// TwinCAT 3 PLC project PLC_
// ProgramVersion: 3.1.4026.24
// libraries:
//   Tc2_EtherCAT, * (Beckhoff Automation GmbH)
//   Tc2_MC2, * (Beckhoff Automation GmbH)
//   Tc2_Standard, * (Beckhoff Automation GmbH)
//   Tc2_SUPS, * (Beckhoff Automation GmbH)
//   Tc2_System, * (Beckhoff Automation GmbH)
//   Tc2_Utilities, * (Beckhoff Automation GmbH)
//   Tc3_McCollisionAvoidance, * (Beckhoff Automation GmbH)
//   Tc3_McCoordinatedMotion, * (Beckhoff Automation GmbH)
//   Tc3_Module, * (Beckhoff Automation GmbH)
// project tree:
//   00_GVLs/ HardwareIO.TcGVL, Parameter_PERSISTENT.TcGVL, GVL.TcGVL, HMI_Mapp.TcGVL
//   01_POUs/ Automatic_POU.TcPOU, Initial_POU.TcPOU, MAIN.TcPOU
//   01_POUs/static/ Device_POU.TcPOU, prgInputMapp.TcPOU, Recipe_POU.TcPOU, Manual_POU.TcPOU, MST_POU.TcPOU, UPS_POU.TcPOU
//   02_Unit/01_Customization/ Ass_DualServo.TcPOU, Ass_LoadPic.TcPOU, Ass_Openbox.TcPOU, Ass_Pallet.TcPOU, Ass_RBStack.TcPOU, Ass_Sealing.TcPOU, Ass_StackComv.TcPOU, Ass_UnloadNG.TcPOU, FB_RollRightAngle.TcPOU, ITF_AutoStructCommand.TcIO, MainControl.TcPOU, ST_HMIitfStructCommandTester.TcDUT, ST_Parameter.TcDUT, ST_SlotData.TcDUT
//   02_Unit/03_Axis/ AXIS_REF_Ext.TcPOU, FB_AxisGeneral.TcPOU, ST_HMIAxieControl.TcDUT, FB_ORG_PositiveEndLessByTouchprobe.TcPOU
//   02_Unit/04_Kuka/ E_KR_AutoExtState.TcDUT, E_CS_Status.TcDUT, RB_KR_PickPlace.TcPOU, RB_KR_Stacking.TcPOU, ST_CS_PickIO.TcDUT, ST_KR_sysIO.TcDUT, ST_KR_stackingIO.TcDUT, ST_CS_sysIO.TcDUT
//   02_Unit/99_Other/ FB_EL3356_0010.TcPOU, FB_RecordValue.TcPOU, F_TrimRightSpace.TcPOU, ST_Inventer.TcDUT, ST_InventerUD.TcDUT, Spacil_FC.TcPOU, ST_Operation.TcDUT
//   02_Unit/00_Alarm/ E_Alarm.TcDUT, E_Warn.TcDUT, ST_AlarmFlag.TcDUT, ST_AlarmItem.TcDUT, U_Alarm.TcDUT
//   / GlobalTextList.TcGTLO, LowTask.TcTTO, PlcTask.TcTTO, RecipeManager.TcRMO (not stored)
//   02_Unit/02_Cylinder kit/ E_CylFault.TcTLEO, E_CylinderType.TcTLEO, FB_CylinderBase.TcPOU, ST_Cylinder.TcDUT, ST_CylinderParameter.TcDUT
//   02_Unit/11_EventLogger/ EventLogger.TcPOU, E_EventType.TcTLEO, ST_Event.TcDUT, UpdateEventTimeWithSystemTime.TcPOU
// real-time tasks:
//   TASK PlcTask: cycle T#1ms, priority 20, ADS port 350
//   TASK Job Task: cycle default, priority 32
//   TASK EipTask: cycle T#10ms, priority 1, ADS port 301
//   TASK LowTask: cycle T#10ms, priority 2, ADS port 351
// motion (NC):
//   TASK NC-Task 1 SAF: cycle T#1ms, priority 4, ADS port 501
//   TASK NC-Task 1 SVB: cycle T#2ms, priority 8, ADS port 511
//   AXIS Axis DualServo1 2 (id 1)
//     Dynamic: Acceleration=70000.1, Deceleration=70000.1, Jerk=1633330
//     Velo: Maximum=4000
//     OtherSettings: AllowMotionCmdToSlave=true
//     encoder EncType=19
//       EncPara: ScaleFactorNumerator=91.44, ScaleFactorDenominator=8388608, ModuloFactor=3657.5, Inverse=true, MaxCount=#xffffffff
//         ActPosCorrection: Enable=true, Time=0.1
//     drive DrvType=16
//       DrvPara: Inverse=true, MaxCount=#xffffffff, DriveControlDWord=#x00020100
//         Analog: VeloReferenz=4000, TorqueSetpointScale=10, ScaleFactorActTorque=0.1
//         TimeComp: TaskDelayCycles=1
//     controller CtrType=1
//       CtrPara: PriorControlFactor=1
//         PosDiffControl: Enable=false
//         Observer: BandWidth=20
//   AXIS Axis DualServo2 3 (id 2)
//     Dynamic: Acceleration=70000.1, Deceleration=70000.1, Jerk=1633330
//     Velo: Maximum=4000
//     OtherSettings: AllowMotionCmdToSlave=true
//     encoder EncType=19
//       EncPara: ScaleFactorNumerator=91.44, ScaleFactorDenominator=8388608, ModuloFactor=3657.5, Inverse=true, MaxCount=#xffffffff
//         ActPosCorrection: Enable=true, Time=0.1
//     drive DrvType=16
//       DrvPara: Inverse=true, MaxCount=#xffffffff, DriveControlDWord=#x00020100
//         Analog: VeloReferenz=4000, TorqueSetpointScale=10, ScaleFactorActTorque=0.1
//         TimeComp: TaskDelayCycles=1
//     controller CtrType=1
//       CtrPara: PriorControlFactor=1
//         PosDiffControl: Enable=false
//         Observer: BandWidth=20
//   AXIS Axis_FlyIn 1 (id 3)
//     Dynamic: Acceleration=28000, Deceleration=28000, Jerk=653333
//     Velo: Maximum=1600
//     PositionAreaControl: Enable=false
//     TargetPosControl: Enable=false
//     OtherSettings: AllowMotionCmdToSlave=true
//     encoder EncType=19
//       EncPara: ScaleFactorNumerator=31.9024, ScaleFactorDenominator=8388608, Inverse=true, MaxCount=#xffffffff
//     drive DrvType=16
//       DrvPara: Inverse=true, MaxCount=#xffffffff, DriveControlDWord=#x00020100
//         Analog: TorqueSetpointScale=10, ScaleFactorActTorque=0.1
//         TimeComp: TaskDelayCycles=1
//     controller CtrType=1
//       CtrPara: PriorControlFactor=1
//         PosDiffControl: Enable=false
//         Observer: BandWidth=20
//   AXIS Axis BoxPullout 4 (id 4)
//     Dynamic: Acceleration=12750, Deceleration=12750, Jerk=154821
//     Velo: FastManual=300, Maximum=1500
//     OtherSettings: AllowMotionCmdToSlave=true
//     encoder EncType=19
//       EncPara: ScaleFactorNumerator=6.2831853, ScaleFactorDenominator=8388608, Inverse=true, MaxCount=#xffffffff
//     drive DrvType=16
//       DrvPara: Inverse=true, MaxCount=#xffffffff, DriveControlDWord=#x00020100
//         Analog: VeloReferenz=1500, TorqueSetpointScale=10, ScaleFactorActTorque=0.1
//         TimeComp: TaskDelayCycles=1
//     controller CtrType=1
//       CtrPara: PriorControlFactor=1
//         Observer: BandWidth=20
//   AXIS Axis load1 5 (id 5)
//     Dynamic: Acceleration=12000, Deceleration=12000, Jerk=90000
//     Velo: RefSearch=300, RefSync=300
//     OtherSettings: AllowMotionCmdToSlave=true
//     encoder EncType=19
//       EncPara: ScaleFactorNumerator=31.41599265359, ScaleFactorDenominator=8388608, ModuloFactor=1005, MaxCount=#xffffffff
//         Inc: RefSearchInverse=true, RefSyncInverse=false
//     drive DrvType=16
//       DrvPara: MaxCount=#xffffffff, DriveControlDWord=#x00020100
//         Analog: TorqueSetpointScale=10, ScaleFactorActTorque=0.1
//         TimeComp: TaskDelayCycles=1
//     controller CtrType=1
//       CtrPara: PriorControlFactor=1
//         PosDiffControl: Enable=false
//         Observer: BandWidth=20
//   AXIS Axis load2 6 (id 6)
//     Dynamic: Acceleration=12000, Deceleration=12000, Jerk=90000
//     Velo: RefSearch=300, RefSync=300
//     OtherSettings: AllowMotionCmdToSlave=true
//     encoder EncType=19
//       EncPara: ScaleFactorNumerator=31.41599265359, ScaleFactorDenominator=8388608, ModuloFactor=1005, Inverse=true, MaxCount=#xffffffff
//         Inc: RefSearchInverse=true, RefSyncInverse=false
//     drive DrvType=16
//       DrvPara: Inverse=true, MaxCount=#xffffffff, DriveControlDWord=#x00020100
//         Analog: TorqueSetpointScale=10, ScaleFactorActTorque=0.1
//         TimeComp: TaskDelayCycles=1
//     controller CtrType=1
//       CtrPara: PriorControlFactor=1
//         PosDiffControl: Enable=false
//         Observer: BandWidth=20
// I/O:
//   DEVICE Device 1 (EtherCAT), AmsNetId 10.200.96.23.2.1
//     Term 1 (EK1200) [EK1200-5000 EtherCAT Power supply (2A E-Bus)]
//       Term 2 (EL1889) [EL1889 16Ch. Dig. Input 24V, 3ms, negative]
//       Term 3 (EL1889) [EL1889 16Ch. Dig. Input 24V, 3ms, negative]
//       Term 4 (EL1889) [EL1889 16Ch. Dig. Input 24V, 3ms, negative]
//       Term 5 (EL1889) [EL1889 16Ch. Dig. Input 24V, 3ms, negative]
//       Term 6 (EL2889) [EL2889 16Ch. Dig. Output 24V, 0.5A, negative]
//       Term 7 (EL2889) [EL2889 16Ch. Dig. Output 24V, 0.5A, negative]
//       Term 8 (EL2889) [EL2889 16Ch. Dig. Output 24V, 0.5A, negative]
//       Term 9 (EL9510) [EL9510 Power supply terminal 10V]
//       Term 10 (EL3356-0010) [EL3356-0010 1Ch. Ana. Input Resistor Bridge Terminal, 24bit, High Precision]
//       Term 11 (EK1110) [EK1110 EtherCAT extension]
//     Drive 12 (MBDLN25BE) [MBDLN25BE]
//     Drive 13 (MCDLN35BE) [MCDLN35BE]
//     Drive 14 (MCDLN35BE) [MCDLN35BE]
//     Drive 15 (MCDLN35BE) [MCDLN35BE]
//     Drive 16 (MBDLN25BE) [MBDLN25BE]
//     Drive 17 (MBDLN25BE) [MBDLN25BE]
//   DEVICE Device 2 (TC3 EIP Scanner), AmsNetId 10.200.96.23.3.1
//     Box 18 (KR CS-Box2) // <INFO> </INFO> <EDS> C:\TwinCAT\3.1\Config\Io\EtherNetIP\KR_CS-Box2 (1).EDS </EDS>
//     Box 19 (KR C5 - EtherNet/IP) // <INFO> </INFO> <EDS> C:\TwinCAT\3.1\Config\Io\EtherNetIP\KRC5EtherNetIP.eds </EDS>
// variable links:
//   NC-Task 1 SAF/Axes/Axis BoxPullout 4 <-> Device 1 (EtherCAT)/Drive 15 (MCDLN35BE)
//     Drive/Inputs/In/nDataIn1 <-> Transmit PDO mapping 1/Following error actual value
//     Drive/Inputs/In/nState1 <-> Transmit PDO mapping 1/Statusword
//     Drive/Inputs/In/nState2 <-> Transmit PDO mapping 1/Statusword @bit 8
//     Drive/Inputs/In/nState4 @bit 1 <-> WcState/InputToggle
//     Drive/Inputs/In/nState4 <-> WcState/WcState
//     Drive/Inputs/In/nState5 <-> Transmit PDO mapping 1/Modes of operation display
//     Drive/Outputs/Out/nCtrl1 <-> Receive PDO mapping 1/Controlword
//     Drive/Outputs/Out/nCtrl2 <-> Receive PDO mapping 1/Controlword @bit 8
//     Drive/Outputs/Out/nCtrl5 <-> Receive PDO mapping 1/Modes of operation
//     Drive/Outputs/Out/nDataOut1 <-> Receive PDO mapping 1/Target position
//     Enc/Inputs/In/nDataIn1 <-> Transmit PDO mapping 1/Position actual value
//     Enc/Inputs/In/nDataIn3 <-> Transmit PDO mapping 1/Touch probe pos1 pos value
//     Enc/Inputs/In/nState4 @bit 1 <-> WcState/InputToggle
//     Enc/Inputs/In/nState4 <-> WcState/WcState
//     Enc/Inputs/In/nState5 <-> Transmit PDO mapping 1/Touch probe status
//     Enc/Inputs/In/nState6 <-> Transmit PDO mapping 1/Touch probe status @bit 8
//     Enc/Outputs/Out/nCtrl5 <-> Receive PDO mapping 1/Touch probe function
//     Enc/Outputs/Out/nCtrl6 <-> Receive PDO mapping 1/Touch probe function @bit 8
//   NC-Task 1 SAF/Axes/Axis DualServo1 2 <-> Device 1 (EtherCAT)/Drive 13 (MCDLN35BE)
//     Drive/Inputs/In/nDataIn1 <-> Transmit PDO mapping 1/Following error actual value
//     Drive/Inputs/In/nState1 <-> Transmit PDO mapping 1/Statusword
//     Drive/Inputs/In/nState2 <-> Transmit PDO mapping 1/Statusword @bit 8
//     Drive/Inputs/In/nState4 @bit 1 <-> WcState/InputToggle
//     Drive/Inputs/In/nState4 <-> WcState/WcState
//     Drive/Inputs/In/nState5 <-> Transmit PDO mapping 1/Modes of operation display
//     Drive/Outputs/Out/nCtrl1 <-> Receive PDO mapping 1/Controlword
//     Drive/Outputs/Out/nCtrl2 <-> Receive PDO mapping 1/Controlword @bit 8
//     Drive/Outputs/Out/nCtrl5 <-> Receive PDO mapping 1/Modes of operation
//     Drive/Outputs/Out/nDataOut1 <-> Receive PDO mapping 1/Target position
//     Enc/Inputs/In/nDataIn1 <-> Transmit PDO mapping 1/Position actual value
//     Enc/Inputs/In/nDataIn3 <-> Transmit PDO mapping 1/Touch probe pos1 pos value
//     Enc/Inputs/In/nState4 @bit 1 <-> WcState/InputToggle
//     Enc/Inputs/In/nState4 <-> WcState/WcState
//     Enc/Inputs/In/nState5 <-> Transmit PDO mapping 1/Touch probe status
//     Enc/Inputs/In/nState6 <-> Transmit PDO mapping 1/Touch probe status @bit 8
//     Enc/Outputs/Out/nCtrl5 <-> Receive PDO mapping 1/Touch probe function
//     Enc/Outputs/Out/nCtrl6 <-> Receive PDO mapping 1/Touch probe function @bit 8
//   NC-Task 1 SAF/Axes/Axis DualServo2 3 <-> Device 1 (EtherCAT)/Drive 14 (MCDLN35BE)
//     Drive/Inputs/In/nDataIn1 <-> Transmit PDO mapping 1/Following error actual value
//     Drive/Inputs/In/nState1 <-> Transmit PDO mapping 1/Statusword
//     Drive/Inputs/In/nState2 <-> Transmit PDO mapping 1/Statusword @bit 8
//     Drive/Inputs/In/nState4 @bit 1 <-> WcState/InputToggle
//     Drive/Inputs/In/nState4 <-> WcState/WcState
//     Drive/Inputs/In/nState5 <-> Transmit PDO mapping 1/Modes of operation display
//     Drive/Outputs/Out/nCtrl1 <-> Receive PDO mapping 1/Controlword
//     Drive/Outputs/Out/nCtrl2 <-> Receive PDO mapping 1/Controlword @bit 8
//     Drive/Outputs/Out/nCtrl5 <-> Receive PDO mapping 1/Modes of operation
//     Drive/Outputs/Out/nDataOut1 <-> Receive PDO mapping 1/Target position
//     Enc/Inputs/In/nDataIn1 <-> Transmit PDO mapping 1/Position actual value
//     Enc/Inputs/In/nDataIn3 <-> Transmit PDO mapping 1/Touch probe pos1 pos value
//     Enc/Inputs/In/nState4 @bit 1 <-> WcState/InputToggle
//     Enc/Inputs/In/nState4 <-> WcState/WcState
//     Enc/Inputs/In/nState5 <-> Transmit PDO mapping 1/Touch probe status
//     Enc/Inputs/In/nState6 <-> Transmit PDO mapping 1/Touch probe status @bit 8
//     Enc/Outputs/Out/nCtrl5 <-> Receive PDO mapping 1/Touch probe function
//     Enc/Outputs/Out/nCtrl6 <-> Receive PDO mapping 1/Touch probe function @bit 8
//   NC-Task 1 SAF/Axes/Axis load1 5 <-> Device 1 (EtherCAT)/Drive 16 (MBDLN25BE)
//     Drive/Inputs/In/nDataIn1 <-> Transmit PDO mapping 1/Following error actual value
//     Drive/Inputs/In/nState1 <-> Transmit PDO mapping 1/Statusword
//     Drive/Inputs/In/nState2 <-> Transmit PDO mapping 1/Statusword @bit 8
//     Drive/Inputs/In/nState4 @bit 1 <-> WcState/InputToggle
//     Drive/Inputs/In/nState4 <-> WcState/WcState
//     Drive/Inputs/In/nState5 <-> Transmit PDO mapping 1/Modes of operation display
//     Drive/Outputs/Out/nCtrl1 <-> Receive PDO mapping 1/Controlword
//     Drive/Outputs/Out/nCtrl2 <-> Receive PDO mapping 1/Controlword @bit 8
//     Drive/Outputs/Out/nCtrl5 <-> Receive PDO mapping 1/Modes of operation
//     Drive/Outputs/Out/nDataOut1 <-> Receive PDO mapping 1/Target position
//     Enc/Inputs/In/nDataIn1 <-> Transmit PDO mapping 1/Position actual value
//     Enc/Inputs/In/nDataIn3 <-> Transmit PDO mapping 1/Touch probe pos1 pos value
//     Enc/Inputs/In/nState4 @bit 1 <-> WcState/InputToggle
//     Enc/Inputs/In/nState4 <-> WcState/WcState
//     Enc/Inputs/In/nState5 <-> Transmit PDO mapping 1/Touch probe status
//     Enc/Inputs/In/nState6 <-> Transmit PDO mapping 1/Touch probe status @bit 8
//     Enc/Outputs/Out/nCtrl5 <-> Receive PDO mapping 1/Touch probe function
//     Enc/Outputs/Out/nCtrl6 <-> Receive PDO mapping 1/Touch probe function @bit 8
//   NC-Task 1 SAF/Axes/Axis load2 6 <-> Device 1 (EtherCAT)/Drive 17 (MBDLN25BE)
//     Drive/Inputs/In/nDataIn1 <-> Transmit PDO mapping 1/Following error actual value
//     Drive/Inputs/In/nState1 <-> Transmit PDO mapping 1/Statusword
//     Drive/Inputs/In/nState2 <-> Transmit PDO mapping 1/Statusword @bit 8
//     Drive/Inputs/In/nState4 @bit 1 <-> WcState/InputToggle
//     Drive/Inputs/In/nState4 <-> WcState/WcState
//     Drive/Inputs/In/nState5 <-> Transmit PDO mapping 1/Modes of operation display
//     Drive/Outputs/Out/nCtrl1 <-> Receive PDO mapping 1/Controlword
//     Drive/Outputs/Out/nCtrl2 <-> Receive PDO mapping 1/Controlword @bit 8
//     Drive/Outputs/Out/nCtrl5 <-> Receive PDO mapping 1/Modes of operation
//     Drive/Outputs/Out/nDataOut1 <-> Receive PDO mapping 1/Target position
//     Enc/Inputs/In/nDataIn1 <-> Transmit PDO mapping 1/Position actual value
//     Enc/Inputs/In/nDataIn3 <-> Transmit PDO mapping 1/Touch probe pos1 pos value
//     Enc/Inputs/In/nState4 @bit 1 <-> WcState/InputToggle
//     Enc/Inputs/In/nState4 <-> WcState/WcState
//     Enc/Inputs/In/nState5 <-> Transmit PDO mapping 1/Touch probe status
//     Enc/Inputs/In/nState6 <-> Transmit PDO mapping 1/Touch probe status @bit 8
//     Enc/Outputs/Out/nCtrl5 <-> Receive PDO mapping 1/Touch probe function
//     Enc/Outputs/Out/nCtrl6 <-> Receive PDO mapping 1/Touch probe function @bit 8
//   NC-Task 1 SAF/Axes/Axis_FlyIn 1 <-> Device 1 (EtherCAT)/Drive 12 (MBDLN25BE)
//     Drive/Inputs/In/nDataIn1 <-> Transmit PDO mapping 1/Following error actual value
//     Drive/Inputs/In/nState1 <-> Transmit PDO mapping 1/Statusword
//     Drive/Inputs/In/nState2 <-> Transmit PDO mapping 1/Statusword @bit 8
//     Drive/Inputs/In/nState4 @bit 1 <-> WcState/InputToggle
//     Drive/Inputs/In/nState4 <-> WcState/WcState
//     Drive/Inputs/In/nState5 <-> Transmit PDO mapping 1/Modes of operation display
//     Drive/Outputs/Out/nCtrl1 <-> Receive PDO mapping 1/Controlword
//     Drive/Outputs/Out/nCtrl2 <-> Receive PDO mapping 1/Controlword @bit 8
//     Drive/Outputs/Out/nCtrl5 <-> Receive PDO mapping 1/Modes of operation
//     Drive/Outputs/Out/nDataOut1 <-> Receive PDO mapping 1/Target position
//     Enc/Inputs/In/nDataIn1 <-> Transmit PDO mapping 1/Position actual value
//     Enc/Inputs/In/nDataIn3 <-> Transmit PDO mapping 1/Touch probe pos1 pos value
//     Enc/Inputs/In/nState4 @bit 1 <-> WcState/InputToggle
//     Enc/Inputs/In/nState4 <-> WcState/WcState
//     Enc/Inputs/In/nState5 <-> Transmit PDO mapping 1/Touch probe status
//     Enc/Inputs/In/nState6 <-> Transmit PDO mapping 1/Touch probe status @bit 8
//     Enc/Outputs/Out/nCtrl5 <-> Receive PDO mapping 1/Touch probe function
//     Enc/Outputs/Out/nCtrl6 <-> Receive PDO mapping 1/Touch probe function @bit 8
//   PLC_/PLC_ Instance <-> Device 1 (EtherCAT)/Drive 12 (MBDLN25BE)
//     PlcTask Inputs/HardwareIO.Axis_FlyIn.DI <-> Transmit PDO mapping 1/Digital inputs
//     PlcTask Inputs/HardwareIO.Axis_FlyIn.DeviceErrorcode <-> Transmit PDO mapping 1/Error code
//     PlcTask Inputs/HardwareIO.Axis_FlyIn.stEcSlaveAmsNetAdr <-> InfoData/AdsAddr
//     PlcTask Inputs/HardwareIO.MainFiledBus[10] <-> InfoData/State
//   PLC_/PLC_ Instance <-> Device 1 (EtherCAT)/Drive 13 (MCDLN35BE)
//     PlcTask Inputs/HardwareIO.Axis_DualServo1.DI <-> Transmit PDO mapping 1/Digital inputs
//     PlcTask Inputs/HardwareIO.Axis_DualServo1.stEcSlaveAmsNetAdr <-> InfoData/AdsAddr
//     PlcTask Inputs/HardwareIO.MainFiledBus[11] <-> InfoData/State
//   PLC_/PLC_ Instance <-> Device 1 (EtherCAT)/Drive 14 (MCDLN35BE)
//     PlcTask Inputs/HardwareIO.Axis_DualServo2.DI <-> Transmit PDO mapping 1/Digital inputs
//     PlcTask Inputs/HardwareIO.Axis_DualServo2.stEcSlaveAmsNetAdr <-> InfoData/AdsAddr
//     PlcTask Inputs/HardwareIO.MainFiledBus[12] <-> InfoData/State
//   PLC_/PLC_ Instance <-> Device 1 (EtherCAT)/Drive 15 (MCDLN35BE)
//     PlcTask Inputs/HardwareIO.Axis_BoxPullOut.DI <-> Transmit PDO mapping 1/Digital inputs
//     PlcTask Inputs/HardwareIO.Axis_BoxPullOut.stEcSlaveAmsNetAdr <-> InfoData/AdsAddr
//     PlcTask Inputs/HardwareIO.MainFiledBus[13] <-> InfoData/State
//   PLC_/PLC_ Instance <-> Device 1 (EtherCAT)/Drive 16 (MBDLN25BE)
//     PlcTask Inputs/HardwareIO.Axis_load1.stEcSlaveAmsNetAdr <-> InfoData/AdsAddr
//     PlcTask Inputs/HardwareIO.MainFiledBus[14] <-> InfoData/State
//   PLC_/PLC_ Instance <-> Device 1 (EtherCAT)/Drive 17 (MBDLN25BE)
//     PlcTask Inputs/HardwareIO.Axis_load2.stEcSlaveAmsNetAdr <-> InfoData/AdsAddr
//     PlcTask Inputs/HardwareIO.MainFiledBus[15] <-> InfoData/State
//   PLC_/PLC_ Instance <-> Device 1 (EtherCAT)/Term 1 (EK1200)/Term 10 (EL3356-0010)
//     PlcTask Inputs/HardwareIO.LoadCell.bWcState <-> WcState/WcState
//     PlcTask Inputs/HardwareIO.LoadCell.rValue_REAL <-> RMB Value (Real)/Value (Real)
//     PlcTask Inputs/HardwareIO.LoadCell.stEcSlaveAmsNetAdr <-> InfoData/AdsAddr
//     PlcTask Inputs/HardwareIO.LoadCell.wState <-> InfoData/State
//     PlcTask Inputs/HardwareIO.LoadCell.wStatus <-> RMB Status/Status
//     PlcTask Outputs/HardwareIO.LoadCell.wControl <-> RMB Control/Ctrl
//   PLC_/PLC_ Instance <-> Device 1 (EtherCAT)/Term 1 (EK1200)/Term 11 (EK1110)
//     PlcTask Inputs/HardwareIO.MainFiledBus[8] <-> InfoData/State
//   PLC_/PLC_ Instance <-> Device 1 (EtherCAT)/Term 1 (EK1200)/Term 2 (EL1889)
//     PlcTask Inputs/HardwareIO.EL1889[1,11] <-> Channel 11/Input
//     PlcTask Inputs/HardwareIO.EL1889[1,12] <-> Channel 12/Input
//     PlcTask Inputs/HardwareIO.EL1889[1,13] <-> Channel 13/Input
//     PlcTask Inputs/HardwareIO.MainFiledBus[0] <-> InfoData/State
//     PlcTask Inputs/HardwareIO.Motor_Blower.iError <-> Channel 4/HardwareIO.Motor_Blower.iError
//     PlcTask Inputs/HardwareIO.Motor_BoxSealBottom_L.iError <-> Channel 1/HardwareIO.Motor_BoxSealBottom_L.iError
//     PlcTask Inputs/HardwareIO.Motor_BoxSealBottom_R.iError <-> Channel 2/HardwareIO.Motor_BoxSealBottom_R.iError
//     PlcTask Inputs/HardwareIO.Motor_shock.iError <-> Channel 3/HardwareIO.Motor_shock.iError
//     PlcTask Inputs/HardwareIO.Roller_Exit.iError <-> Channel 10/HardwareIO.Roller_Exit.iError
//     PlcTask Inputs/HardwareIO.Roller_LoadcellIn.iError <-> Channel 6/HardwareIO.Roller_LoadcellIn.iError
//     PlcTask Inputs/HardwareIO.Roller_LoadcellOut.iError <-> Channel 7/HardwareIO.Roller_LoadcellOut.iError
//     PlcTask Inputs/HardwareIO.Roller_LoadcellUD.iError <-> Channel 8/HardwareIO.Roller_LoadcellUD.iError
//     PlcTask Inputs/HardwareIO.Roller_Purge.iError <-> Channel 9/HardwareIO.Roller_Purge.iError
//     PlcTask Inputs/HardwareIO.Sen_AxisBoxORG <-> Channel 14/HardwareIO.Sen_AxisBoxORG
//     PlcTask Inputs/HardwareIO.Sen_AxisLoad1ORG <-> Channel 15/HardwareIO.Sen_AxisLoad1ORG
//     PlcTask Inputs/HardwareIO.Sen_AxisLoad2ORG <-> Channel 16/HardwareIO.Sen_AxisLoad2ORG
//     PlcTask Inputs/HardwareIO.Sen_BeltLoadOut <-> Channel 5/HardwareIO.Sen_BeltLoadOut
//   PLC_/PLC_ Instance <-> Device 1 (EtherCAT)/Term 1 (EK1200)/Term 3 (EL1889)
//     PlcTask Inputs/HardwareIO.Cyl_Axis90.iEndSensor <-> Channel 7/HardwareIO.Cyl_Axis90.iEndSensor
//     PlcTask Inputs/HardwareIO.Cyl_Axis90.iOriginSensor <-> Channel 8/HardwareIO.Cyl_Axis90.iOriginSensor
//     PlcTask Inputs/HardwareIO.Cyl_AxisBottom.iEndSensor <-> Channel 10/HardwareIO.Cyl_AxisBottom.iEndSensor
//     PlcTask Inputs/HardwareIO.Cyl_AxisBottom.iOriginSensor <-> Channel 11/HardwareIO.Cyl_AxisBottom.iOriginSensor
//     PlcTask Inputs/HardwareIO.Cyl_AxisBoxCatch.iEndSensor <-> Channel 4/HardwareIO.Cyl_AxisBoxCatch.iEndSensor
//     PlcTask Inputs/HardwareIO.Cyl_AxisBoxCatch.iOriginSensor <-> Channel 5/HardwareIO.Cyl_AxisBoxCatch.iOriginSensor
//     PlcTask Inputs/HardwareIO.Cyl_BeltBottom.iEndSensor <-> Channel 12/HardwareIO.Cyl_BeltBottom.iEndSensor
//     PlcTask Inputs/HardwareIO.Cyl_BeltBottom.iOriginSensor <-> Channel 13/HardwareIO.Cyl_BeltBottom.iOriginSensor
//     PlcTask Inputs/HardwareIO.Cyl_BoxSidePitch.iEndSensor <-> Channel 3/HardwareIO.Cyl_BoxSidePitch.iEndSensor
//     PlcTask Inputs/HardwareIO.Cyl_BoxSidePitch.iOriginSensor <-> Channel 2/HardwareIO.Cyl_BoxSidePitch.iOriginSensor
//     PlcTask Inputs/HardwareIO.MainFiledBus[1] <-> InfoData/State
//     PlcTask Inputs/HardwareIO.Sen_Axis90Vacumm <-> Channel 9/HardwareIO.Sen_Axis90Vacumm
//     PlcTask Inputs/HardwareIO.Sen_AxisBoxCatchVacumm <-> Channel 6/HardwareIO.Sen_AxisBoxCatchVacumm
//     PlcTask Inputs/HardwareIO.Sen_BoxsideFeed <-> Channel 1/HardwareIO.Sen_BoxsideFeed
//     PlcTask Inputs/HardwareIO.Sen_NGLoadOut <-> Channel 16/HardwareIO.Sen_NGLoadOut
//     PlcTask Inputs/HardwareIO.Sen_TFLoadIn <-> Channel 15/HardwareIO.Sen_TFLoadIn
//     PlcTask Inputs/HardwareIO.Sen_UnloadLoadPos <-> Channel 14/HardwareIO.Sen_UnloadLoadPos
//   PLC_/PLC_ Instance <-> Device 1 (EtherCAT)/Term 1 (EK1200)/Term 4 (EL1889)
//     PlcTask Inputs/HardwareIO.Bundling_ErrorSignal <-> Channel 10/HardwareIO.Bundling_ErrorSignal
//     PlcTask Inputs/HardwareIO.Cyl_NGPurge.iEndSensor <-> Channel 1/HardwareIO.Cyl_NGPurge.iEndSensor
//     PlcTask Inputs/HardwareIO.Cyl_ShockStop.iOriginSensor <-> Channel 3/HardwareIO.Cyl_ShockStop.iEndSensor
//     PlcTask Inputs/HardwareIO.Cyl_StackUD.iEndSensor <-> Channel 5/HardwareIO.Cyl_StackUD.iEndSensor
//     PlcTask Inputs/HardwareIO.Cyl_StackUD.iOriginSensor <-> Channel 6/HardwareIO.Cyl_StackUD.iOriginSensor
//     PlcTask Inputs/HardwareIO.MainFiledBus[2] <-> InfoData/State
//     PlcTask Inputs/HardwareIO.PB_EMG <-> Channel 13/HardwareIO.PB_EMG
//     PlcTask Inputs/HardwareIO.PB_Start <-> Channel 11/HardwareIO.PB_Start
//     PlcTask Inputs/HardwareIO.PB_Stop <-> Channel 12/HardwareIO.PB_Stop
//     PlcTask Inputs/HardwareIO.Sen_ExitBoxCheck <-> Channel 8/HardwareIO.Sen_ExitBoxCheck
//     PlcTask Inputs/HardwareIO.Sen_ExitComvStop <-> Channel 9/HardwareIO.Sen_ExitComvStop
//     PlcTask Inputs/HardwareIO.Sen_ShockPos <-> Channel 2/HardwareIO.Sen_ShockPos
//     PlcTask Inputs/HardwareIO.Sen_StackComvStop <-> Channel 4/HardwareIO.Sen_StackComvStop
//     PlcTask Inputs/HardwareIO.Sen_StackUDVacumm <-> Channel 7/HardwareIO.Sen_StackUDVacumm
//     PlcTask Inputs/HardwareIO.WindowsSafe[1] <-> Channel 14/HardwareIO.WindowsSafe[1]
//     PlcTask Inputs/HardwareIO.WindowsSafe[2] <-> Channel 15/HardwareIO.WindowsSafe[2]
//     PlcTask Inputs/HardwareIO.WindowsSafe[3] <-> Channel 16/HardwareIO.WindowsSafe[3]
//   PLC_/PLC_ Instance <-> Device 1 (EtherCAT)/Term 1 (EK1200)/Term 5 (EL1889)
//     PlcTask Inputs/HardwareIO.Air_Signal <-> Channel 6/HardwareIO.Air_Signal
//     PlcTask Inputs/HardwareIO.Cyl_BoxSideBottom.iEndSensor <-> Channel 8/HardwareIO.Cyl_BoxSideBottom.iEndSensor
//     PlcTask Inputs/HardwareIO.Cyl_BoxSideBottom.iOriginSensor <-> Channel 9/HardwareIO.Cyl_BoxSideBottom.iOriginSensor
//     PlcTask Inputs/HardwareIO.Cyl_UnloadDef.iEndSensor <-> Channel 15/HardwareIO.Cyl_UnloadDef.iEndSensor
//     PlcTask Inputs/HardwareIO.Cyl_UnloadDef.iOriginSensor <-> Channel 16/HardwareIO.Cyl_UnloadDef.iOriginSensor
//     PlcTask Inputs/HardwareIO.MainFiledBus[3] <-> InfoData/State
//     PlcTask Inputs/HardwareIO.Motor_Stack.iError <-> Channel 13/HardwareIO.Motor_Stack.iError
//     PlcTask Inputs/HardwareIO.Roller_LoadcellUD.iHighPos <-> Channel 11/HardwareIO.Roller_LoadcellUD.iHighPos
//     PlcTask Inputs/HardwareIO.Roller_LoadcellUD.iLowPos <-> Channel 12/HardwareIO.Roller_LoadcellUD.iLowPos
//     PlcTask Inputs/HardwareIO.Sen_BeltLoadIn <-> Channel 10/HardwareIO.Sen_BeltLoadIn
//     PlcTask Inputs/HardwareIO.Sen_BoxsideStorageMaterial <-> Channel 5/HardwareIO.Sen_BoxsideStorageMaterial
//     PlcTask Inputs/HardwareIO.Sen_ExitLoadIn <-> Channel 7/HardwareIO.Sen_ExitLoadIn
//     PlcTask Inputs/HardwareIO.Swtich_PassFeet <-> Channel 4/HardwareIO.Swtich_PassFeet
//     PlcTask Inputs/HardwareIO.TemperatureHigh <-> Channel 14/HardwareIO.TemperatureHigh
//     PlcTask Inputs/HardwareIO.WindowsSafe[4] <-> Channel 1/HardwareIO.WindowsSafe[4]
//     PlcTask Inputs/HardwareIO.WindowsSafe[5] <-> Channel 2/HardwareIO.WindowsSafe[5]
//     PlcTask Inputs/HardwareIO.WindowsSafe[6] <-> Channel 3/HardwareIO.WindowsSafe[6]
//   PLC_/PLC_ Instance <-> Device 1 (EtherCAT)/Term 1 (EK1200)/Term 6 (EL2889)
//     PlcTask Inputs/HardwareIO.MainFiledBus[4] <-> InfoData/State
//     PlcTask Outputs/HardwareIO.Cyl_AxisBoxCatch.qExtendCoil <-> Channel 16/HardwareIO.Cyl_AxisBoxCatch.qExtendCoil
//     PlcTask Outputs/HardwareIO.Cyl_BoxSidePitch.qExtendCoil <-> Channel 15/HardwareIO.Cyl_BoxSidePitch.qExtendCoil
//     PlcTask Outputs/HardwareIO.Motor_Blower.qRun <-> Channel 8/HardwareIO.Motor_Blower.qRun
//     PlcTask Outputs/HardwareIO.Motor_BoxSealBottom_L.qRun <-> Channel 5/HardwareIO.Motor_BoxSealBottom_L.qRun
//     PlcTask Outputs/HardwareIO.Motor_BoxSealBottom_R.qRun <-> Channel 6/HardwareIO.Motor_BoxSealBottom_R.qRun
//     PlcTask Outputs/HardwareIO.Motor_LoadIn.qRun <-> Channel 1/HardwareIO.Motor_LoadIn.qRun
//     PlcTask Outputs/HardwareIO.Motor_LoadPurge1.qRun <-> Channel 2/HardwareIO.Motor_LoadPurge1.qRun
//     PlcTask Outputs/HardwareIO.Motor_LoadPurge2.qRun <-> Channel 3/HardwareIO.Motor_LoadPurge2.qRun
//     PlcTask Outputs/HardwareIO.Motor_Stack.qRun <-> Channel 4/HardwareIO.Motor_Stack.qRun
//     PlcTask Outputs/HardwareIO.Motor_shock.qRun <-> Channel 7/HardwareIO.Motor_shock.qRun
//     PlcTask Outputs/HardwareIO.Roller_Exit.qRun <-> Channel 14/HardwareIO.Roller_Exit.qRun
//     PlcTask Outputs/HardwareIO.Roller_LoadcellIn.qRun <-> Channel 9/HardwareIO.Roller_LoadcellIn.qRun
//     PlcTask Outputs/HardwareIO.Roller_LoadcellOut.qRun <-> Channel 10/HardwareIO.Roller_LoadcellOut.qRun
//     PlcTask Outputs/HardwareIO.Roller_LoadcellUD.qRun <-> Channel 11/HardwareIO.Roller_LoadcellUD.qRun
//     PlcTask Outputs/HardwareIO.Roller_LoadcellUD.qSign <-> Channel 12/HardwareIO.Roller_LoadcellUD.qSign
//     PlcTask Outputs/HardwareIO.Roller_Purge.qRun <-> Channel 13/HardwareIO.Roller_Purge.qRun
//   PLC_/PLC_ Instance <-> Device 1 (EtherCAT)/Term 1 (EK1200)/Term 7 (EL2889)
//     PlcTask Inputs/HardwareIO.MainFiledBus[5] <-> InfoData/State
//     PlcTask Outputs/HardwareIO.Cyl_Axis90.qExtendCoil <-> Channel 1/HardwareIO.Cyl_Axis90.qExtendCoil
//     PlcTask Outputs/HardwareIO.Cyl_AxisBottom.qExtendCoil <-> Channel 2/HardwareIO.Cyl_AxisBottom.qExtendCoil
//     PlcTask Outputs/HardwareIO.Cyl_BeltBottom.qExtendCoil <-> Channel 5/HardwareIO.Cyl_BeltBottom.qExtendCoil
//     PlcTask Outputs/HardwareIO.Cyl_BoxSideBottom.qExtendCoil <-> Channel 6/HardwareIO.Cyl_BoxSideBottom.qExtendCoil
//     PlcTask Outputs/HardwareIO.Cyl_ExitClip.qExtendCoil <-> Channel 10/HardwareIO.Cyl_ExitClip.qExtendCoil
//     PlcTask Outputs/HardwareIO.Cyl_ExitStopper.qExtendCoil <-> Channel 11/HardwareIO.Cyl_ExitStopper.qExtendCoil
//     PlcTask Outputs/HardwareIO.Cyl_FlyIn_Pass <-> Channel 13/HardwareIO.Cyl_FlyIn_Pass
//     PlcTask Outputs/HardwareIO.Cyl_ShockStop.qExtendCoil <-> Channel 7/HardwareIO.Cyl_ShockStop.qExtendCoil
//     PlcTask Outputs/HardwareIO.Cyl_StackUD.qExtendCoil <-> Channel 8/HardwareIO.Cyl_StackUD.qExtendCoil
//     PlcTask Outputs/HardwareIO.Light_BZ <-> Channel 14/HardwareIO.Light_BZ
//     PlcTask Outputs/HardwareIO.Light_Red <-> Channel 15/HardwareIO.Light_Red
//     PlcTask Outputs/HardwareIO.Light_Yellow <-> Channel 16/HardwareIO.Light_Yellow
//     PlcTask Outputs/HardwareIO.Vacm_Axis90 <-> Channel 4/HardwareIO.Vacm_Axis90
//     PlcTask Outputs/HardwareIO.Vacm_AxisCatchBox <-> Channel 3/HardwareIO.Vacm_AxisCatchBox
//     PlcTask Outputs/HardwareIO.Vacm_StackUD <-> Channel 9/HardwareIO.Vacm_StackUD
//   PLC_/PLC_ Instance <-> Device 1 (EtherCAT)/Term 1 (EK1200)/Term 8 (EL2889)
//     PlcTask Inputs/HardwareIO.MainFiledBus[6] <-> InfoData/State
//     PlcTask Outputs/HardwareIO.Bundling_yPause <-> Channel 11/HardwareIO.Bundling_yPause
//     PlcTask Outputs/HardwareIO.Cyl_BeltBottomSup.qExtendCoil <-> Channel 5/HardwareIO.Cyl_BeltBottomSup.qExtendCoil
//     PlcTask Outputs/HardwareIO.Cyl_NGPurge.qExtendCoil <-> Channel 6/HardwareIO.Cyl_NGPurge.qExtendCoil
//     PlcTask Outputs/HardwareIO.Cyl_UnloadDef.qExtendCoil <-> Channel 9/HardwareIO.Cyl_UnloadDef.qExtendCoil
//     PlcTask Outputs/HardwareIO.EL2889[3,{12..16}] <-> Channel {12..16}/Output  (5 links)
//     PlcTask Outputs/HardwareIO.ElectronicBoxLight <-> Channel 10/HardwareIO.ElectronicBoxLight
//     PlcTask Outputs/HardwareIO.Light_Green <-> Channel 1/HardwareIO.Light_Green
//     PlcTask Outputs/HardwareIO.Motor_shock.qSign <-> Channel 7/HardwareIO.Motor_shock.qSign
//     PlcTask Outputs/HardwareIO.TemperatureFans <-> Channel 8/HardwareIO.TemperatureFans
//   PLC_/PLC_ Instance <-> Device 1 (EtherCAT)/Term 1 (EK1200)/Term 9 (EL9510)
//     PlcTask Inputs/HardwareIO.MainFiledBus[7] <-> InfoData/State
//   PLC_/PLC_ Instance <-> Device 2 (TC3 EIP Scanner)/Box 18 (KR CS-Box2)
//     PlcTask Inputs/HardwareIO.RB_CS.aryEIPInput <-> Connection 1 (Input/Output)/Inputs/Input Data
//     PlcTask Inputs/HardwareIO.RB_CS.aryEIPInput @bit {16..1008 step 16} <-> Connection 1 (Input/Output)/Inputs/Input Data_{1..63}  (63 links)
//     PlcTask Inputs/HardwareIO.RB_CS.state <-> Inputs/State
//     PlcTask Outputs/HardwareIO.RB_CS.aryEIPOutput <-> Connection 1 (Input/Output)/Outputs/Output Data
//     PlcTask Outputs/HardwareIO.RB_CS.aryEIPOutput @bit {16..1008 step 16} <-> Connection 1 (Input/Output)/Outputs/Output Data_{1..63}  (63 links)
//   PLC_/PLC_ Instance <-> Device 2 (TC3 EIP Scanner)/Box 19 (KR C5 - EtherNet/IP)
//     PlcTask Inputs/HardwareIO.RB_KR.aryEIPInput <-> Connection 2 (Input/Output)/Inputs/noname0_arrBYTE
//     PlcTask Inputs/HardwareIO.RB_KR.state <-> Inputs/State
//     PlcTask Outputs/HardwareIO.RB_KR.aryEIPOutput <-> Connection 2 (Input/Output)/Outputs/noname0_arrBYTE[0]
//     PlcTask Outputs/HardwareIO.RB_KR.aryEIPOutput @bit {8..1016 step 8} <-> Connection 2 (Input/Output)/Outputs/noname0_arrBYTE[{1..127}]  (127 links)
//   PLC_/PLC_ Instance <-> NC-Task 1 SAF/Axes/Axis BoxPullout 4
//     PlcTask Inputs/HardwareIO.Axis_BoxPullOut.NcToPlc <-> Outputs/ToPlc
//     PlcTask Outputs/HardwareIO.Axis_BoxPullOut.PlcToNc <-> Inputs/FromPlc
//   PLC_/PLC_ Instance <-> NC-Task 1 SAF/Axes/Axis DualServo1 2
//     PlcTask Inputs/HardwareIO.Axis_DualServo1.NcToPlc <-> Outputs/ToPlc
//     PlcTask Outputs/HardwareIO.Axis_DualServo1.PlcToNc <-> Inputs/FromPlc
//   PLC_/PLC_ Instance <-> NC-Task 1 SAF/Axes/Axis DualServo2 3
//     PlcTask Inputs/HardwareIO.Axis_DualServo2.NcToPlc <-> Outputs/ToPlc
//     PlcTask Outputs/HardwareIO.Axis_DualServo2.PlcToNc <-> Inputs/FromPlc
//   PLC_/PLC_ Instance <-> NC-Task 1 SAF/Axes/Axis load1 5
//     PlcTask Inputs/HardwareIO.Axis_load1.NcToPlc <-> Outputs/ToPlc
//     PlcTask Outputs/HardwareIO.Axis_load1.PlcToNc <-> Inputs/FromPlc
//   PLC_/PLC_ Instance <-> NC-Task 1 SAF/Axes/Axis load2 6
//     PlcTask Inputs/HardwareIO.Axis_load2.NcToPlc <-> Outputs/ToPlc
//     PlcTask Outputs/HardwareIO.Axis_load2.PlcToNc <-> Inputs/FromPlc
//   PLC_/PLC_ Instance <-> NC-Task 1 SAF/Axes/Axis_FlyIn 1
//     PlcTask Inputs/HardwareIO.Axis_FlyIn.NcToPlc <-> Outputs/ToPlc
//     PlcTask Outputs/HardwareIO.Axis_FlyIn.PlcToNc <-> Inputs/FromPlc
//   PLC_/PLC_ Instance <-> NC-Task 1 SAF/Objects/Group1 (CA Group)
//     PlcTask Inputs/GVL.DualGroupRef.NcToPlc <-> Group Outputs/ToPLC
//     PlcTask Outputs/GVL.DualGroupRef.PlcToNc <-> Group Inputs/FromPLC

CONFIGURATION PLC_
    RESOURCE PLC ON TwinCAT3
        TASK LowTask(INTERVAL := T#10ms, PRIORITY := 2);
        TASK PlcTask(INTERVAL := T#1ms, PRIORITY := 20);
        PROGRAM Recipe_POU WITH LowTask : Recipe_POU;
        PROGRAM prgInputMapp WITH PlcTask : prgInputMapp;
        PROGRAM Device_POU WITH PlcTask : Device_POU;
        PROGRAM MST_POU WITH PlcTask : MST_POU;
        PROGRAM MAIN WITH PlcTask : MAIN;
        PROGRAM UPS_POU WITH PlcTask : UPS_POU;
    END_RESOURCE
END_CONFIGURATION

// ---- 02_Unit/01_Customization/ST_HMIitfStructCommandTester.TcDUT
TYPE ST_HMIitfStructCommandTester :
STRUCT
	bInitial			:BOOL;
	bInitialTest		:BOOL;
	bProcess			:BOOL;
	bProcessHaltMode	:BOOL;
	bProcessHaltStep	:BOOL;
	bCmdFeedback		:BOOL;
	
	
	
	
END_STRUCT
END_TYPE

// ---- 02_Unit/03_Axis/ST_HMIAxieControl.TcDUT
TYPE ST_HMIAxieControl :
STRUCT
	strStatus	:STRING(30);
	bServoSwitch,bORG,bAbsPos,bINCPos,bJogF,bJogB,bStop,bReset,bSupp1,bSupp2:BOOL;
	CommandAddres	, CommandVelo ,ORGOffset	:REAL;
	moniDI										:UDINT;
	moniDeviceErrorCode							:WORD;
	bMoniReady,bMoniDeviceError	,bMoniHomed,bMoniConpled,bMoniControlLoopClosed				:BOOL;

END_STRUCT
END_TYPE

// ---- 02_Unit/04_Kuka/E_KR_AutoExtState.TcDUT
{attribute 'strict'}
TYPE E_KR_AutoExtState :
(
    Idle := 0,

    CheckReady,
    MoveEnableOn,
    DrivesOnPulse,
    WaitDrivesReady,

    WaitPgnoReq,
    RetryDrivesOnPulse,

    SetProgramNo,
    ExtStartPulse,
    WaitProgramActive,

    Running,
    Finish,

    Error
);
END_TYPE

// ---- 02_Unit/04_Kuka/E_CS_Status.TcDUT
{attribute 'strict'}
TYPE E_CS_Status :
(
    Offline := 0,
	Idle,
	DriveReady,
    ReadyToWork,
    Pou_Runing,
    Pou_Run_Pause,
    Pou_Run_Down,
	EStop,
    Error,
	LessHome,
	StopMess,
	LocalControl,
	DriverOn
);
END_TYPE

// ---- 02_Unit/04_Kuka/ST_CS_PickIO.TcDUT
TYPE ST_CS_PickIO :
STRUCT
    // PLC -> KRC
 	cmd_bBoxInPos			:BOOL;		//紙箱到定位      
	cmd_bPartInPos			:BOOL;		//part到定位
	cmd_wLayer				:BYTE;
	cmd_wIndex				:BYTE;
	cmd_Velo				: BYTE;
    // KRC -> PLC
  	fb_bPacking			:BOOL;		//取料中      
	fb_bPackFinish		:BOOL;		//取料完成
	fb_putting			:BOOL;		//裝箱中
	fb_PutFinish		:BOOL;		//裝箱完成
	fb_PackLayer		:BYTE;		//已裝填層
	fb_Velo				:BYTE;
	fb_wIndex			:BYTE;
END_STRUCT               		
END_TYPE

// ---- 02_Unit/04_Kuka/ST_KR_sysIO.TcDUT
TYPE ST_KR_sysIO :
STRUCT
    // PLC -> KRC
    qDRIVES_ON       : BOOL;   // PLC -> KRC, $DRIVES_ON
    qDRIVES_OFF      : BOOL;   // PLC -> KRC, $DRIVES_OFF
    qMOVE_ENABLE     : BOOL;   // PLC -> KRC, $MOVE_ENABLE
    qCONF_MESS       : BOOL;   // PLC -> KRC, $CONF_MESS
    qEXT_START       : BOOL;   // PLC -> KRC, $EXT_START
    qPGNO            : BYTE;   // PLC -> KRC, program number
    qPGNO_VALID      : BOOL;   // PLC -> KRC, $PGNO_VALID
    // KRC -> PLC
    iEXT_CONTROL     : BOOL;   // KRC -> PLC, $EXT
    iCONTROL_READY   : BOOL;   // KRC -> PLC, control ready
    iSTOP_MESS       : BOOL;   // KRC -> PLC, $STOPMESS
    iDRIVES_READY    : BOOL;   // KRC -> PLC, drives ready
    iPGNO_REQ        : BOOL;   // KRC -> PLC, request program number
    iRobotHomePos    : BOOL;   // KRC -> PLC, $IN_HOME
    iRobotRunning    : BOOL;   // KRC -> PLC, robot running / $PRO_ACT
END_STRUCT               		
END_TYPE

// ---- 02_Unit/04_Kuka/ST_KR_stackingIO.TcDUT
TYPE ST_KR_stackingIO :
STRUCT
	cmd_bPallet_AllowPut		:BOOL;	//棧板_棧板允許堆疊
	cmd_bReady					:BOOL;	//棧板_預約
	cmd_bCount0					:BOOL;		//棧板_歸零
	cmd_bFence					:BOOL;		//棧板_光柵 
	cmd_wSize_length			:INT;	
	cmd_wSize_width				:INT;
	cmd_wSize_height			:INT;
	cmd_wLayer_No				:BYTE;
	cmd_bPartInPos				:BOOL;
	cmd_bSetting2Box			:BOOL;
	cmd_wIndex					:BYTE;
	cmd_Velo					: BYTE;
////////////////////////////////////////////////////	
	fb_wPartNo					:INT;
	fb_bPickFinish				:BOOL;
	fb_bWorking				:BOOL;
	fb_bPalletFinish			:BOOL;
	fb_bPalletInPos			:BOOL;
	fb_wIndex					:BYTE;
	fb_wProNo					:BYTE;
	fb_bError				:ARRAY [0..7]OF BOOL;
END_STRUCT
END_TYPE

// ---- 02_Unit/04_Kuka/ST_CS_sysIO.TcDUT
TYPE ST_CS_sysIO :
STRUCT
    // PLC -> KRC
	qSTOP		: BOOL;		//停止     
	qSTART		: BOOL;     //開始     
	qPAUSE		: BOOL;     //暫停     
	qCONTINUE	: BOOL;     //繼續     
	qRESET		: BOOL;     //停止並卸載  
	qENABLE		: BOOL;     //激活scara
	qPGNO       : BYTE;     //AppID0 
	qACKNOWLEDGEMSG	: BOOL; //確認消息   
	qOVERRIDE		: BOOL; //程序倍率   

    // KRC -> PLC
    iREADY           : BOOL;   // 系統就緒   
    iRUNNING         : BOOL;   // 運行中    
    iPAUSED          : BOOL;   // 已暫停    
    iSTOPPED         : BOOL;   // 已停止    
    iERROR           : BOOL;   // 程序錯誤   
    iSAFEGURAD_ON    : BOOL;   // 安全門已打開 
    iESTOP_ON        : BOOL;   // 緊急停止已按下
	iSERROR				: BOOL;
	iWARING             : BOOL;
	iENABLED            : BOOL;
	iACKNOWLEDGED       : BOOL;
	iERROR_CODE         : BOOL;
	iOVER_RIDE_OUT      : BOOL;
	iHome_Pos			:BOOL;
	iEXT_CONTROL		:BOOL;
END_STRUCT               		
END_TYPE

// ---- 02_Unit/99_Other/ST_Inventer.TcDUT
TYPE ST_Inventer :			//馬達 
STRUCT
	qRun			AT %Q*:BOOL;
	qSign			AT %Q*:BOOL;
	qErrorReset		AT %Q*:BOOL;
	iError			AT %I*:BOOL;	
END_STRUCT
END_TYPE

// ---- 02_Unit/99_Other/ST_InventerUD.TcDUT
TYPE ST_InventerUD EXTENDS ST_Inventer :
STRUCT
	iLowPos			AT %I*:BOOL;		//前往低點位 
	iHighPos		AT %I*:BOOL;		//前往高點位 
END_STRUCT
END_TYPE

// ---- 02_Unit/00_Alarm/E_Alarm.TcDUT
{attribute 'qualified_only'}
{attribute 'strict'}
{attribute 'to_string'}
TYPE E_Alarm :
(
	AL000,
	AL001,
	AL002,
	AL003,
	AL004,
	AL005,
	AL006,
	AL007,
	AL008,
	AL009,
	AL010,
	AL011,
	AL012,
	AL013,
	AL014,
	AL015,
	AL016,
	AL017,
	AL018,
	AL019,
	AL020,
	AL021,
	AL022,
	AL023,
	AL024,
	AL025,
	AL026,
	AL027,
	AL028,
	AL029,
	AL030,
	AL031,
	AL032,
	AL033,
	AL034,
	AL035,
	AL036,
	AL037,
	AL038,
	AL039,
	AL040,
	AL041,
	AL042,
	AL043,
	AL044,
	AL045,
	AL046,
	AL047,
	AL048,
	AL049,
	AL050,
	AL051,
	AL052,
	AL053,
	AL054,
	AL055,
	AL056,
	AL057,
	AL058,
	AL059,
	AL060,
	AL061,
	AL062,
	AL063,
	AL064,
	AL065,
	AL066,
	AL067,
	AL068,
	AL069,
	AL070,
	AL071,
	AL072,
	AL073,
	AL074,
	AL075,
	AL076,
	AL077,
	AL078,
	AL079,
	AL080,
	AL081,
	AL082,
	AL083,
	AL084,
	AL085,
	AL086,
	AL087,
	AL088,
	AL089,
	AL090,
	AL091,
	AL092,
	AL093,
	AL094,
	AL095,
	AL096,
	AL097,
	AL098,
	AL099,
	AL100,
	AL101,
	AL102,
	AL103,
	AL104,
	AL105,
	AL106,
	AL107,
	AL108,
	AL109,
	AL110,
	AL111,
	AL112,
	AL113,
	AL114,
	AL115,
	AL116,
	AL117,
	AL118,
	AL119,
	AL120,
	AL121,
	AL122,
	AL123,
	AL124,
	AL125,
	AL126,
	AL127,
	AL128,
	AL129,
	AL130,
	AL131,
	AL132,
	AL133,
	AL134,
	AL135,
	AL136,
	AL137,
	AL138,
	AL139,
	AL140,
	AL141,
	AL142,
	AL143,
	AL144,
	AL145,
	AL146,
	AL147,
	AL148,
	AL149,
	AL150,
	AL151,
	AL152,
	AL153,
	AL154,
	AL155,
	AL156,
	AL157,
	AL158,
	AL159,
	AL160,
	AL161,
	AL162,
	AL163,
	AL164,
	AL165,
	AL166,
	AL167,
	AL168,
	AL169,
	AL170,
	AL171,
	AL172,
	AL173,
	AL174,
	AL175,
	AL176,
	AL177,
	AL178,
	AL179,
	AL180,
	AL181,
	AL182,
	AL183,
	AL184,
	AL185,
	AL186,
	AL187,
	AL188,
	AL189,
	AL190,
	AL191,
	AL192,
	AL193,
	AL194,
	AL195,
	AL196,
	AL197,
	AL198,
	AL199,
	AL200,
	AL201,
	AL202,
	AL203,
	AL204,
	AL205,
	AL206,
	AL207,
	AL208,
	AL209,
	AL210,
	AL211,
	AL212,
	AL213,
	AL214,
	AL215,
	AL216,
	AL217,
	AL218,
	AL219,
	AL220,
	AL221,
	AL222,
	AL223,
	AL224,
	AL225,
	AL226,
	AL227,
	AL228,
	AL229,
	AL230,
	AL231,
	AL232,
	AL233,
	AL234,
	AL235,
	AL236,
	AL237,
	AL238,
	AL239,
	AL240,
	AL241,
	AL242,
	AL243,
	AL244,
	AL245,
	AL246,
	AL247,
	AL248,
	AL249,
	AL250,
	AL251,
	AL252,
	AL253,
	AL254,
	AL255,
	AL256,
	AL257,
	AL258,
	AL259,
	AL260,
	AL261,
	AL262,
	AL263,
	AL264,
	AL265,
	AL266,
	AL267,
	AL268,
	AL269,
	AL270,
	AL271,
	AL272,
	AL273,
	AL274,
	AL275,
	AL276,
	AL277,
	AL278,
	AL279,
	AL280,
	AL281,
	AL282,
	AL283,
	AL284,
	AL285,
	AL286,
	AL287,
	AL288,
	AL289,
	AL290,
	AL291,
	AL292,
	AL293,
	AL294,
	AL295,
	AL296,
	AL297,
	AL298,
	AL299,
	AL300,
	AL301,
	AL302,
	AL303,
	AL304,
	AL305,
	AL306,
	AL307,
	AL308,
	AL309,
	AL310,
	AL311,
	AL312,
	AL313,
	AL314,
	AL315,
	AL316,
	AL317,
	AL318,
	AL319,
	AL320,
	AL321,
	AL322,
	AL323,
	AL324,
	AL325,
	AL326,
	AL327,
	AL328,
	AL329,
	AL330,
	AL331,
	AL332,
	AL333,
	AL334,
	AL335,
	AL336,
	AL337,
	AL338,
	AL339,
	AL340,
	AL341,
	AL342,
	AL343,
	AL344,
	AL345,
	AL346,
	AL347,
	AL348,
	AL349,
	AL350,
	AL351,
	AL352,
	AL353,
	AL354,
	AL355,
	AL356,
	AL357,
	AL358,
	AL359,
	AL360,
	AL361,
	AL362,
	AL363,
	AL364,
	AL365,
	AL366,
	AL367,
	AL368,
	AL369,
	AL370,
	AL371,
	AL372,
	AL373,
	AL374,
	AL375,
	AL376,
	AL377,
	AL378,
	AL379,
	AL380,
	AL381,
	AL382,  
	AL383,
	AL384,
	AL385,
	AL386,
	AL387,
	AL388,
	AL389,  
	AL390,
	AL391,
	AL392,
	AL393,
	AL394,
	AL395,
	AL396,
	AL397,
	AL398,
	AL399,
	AL400,//B槽主軸伺服馬達_軸錯誤異常   
	AL401,//B槽清洗內罩升降1馬達_軸錯誤異常
	AL402,//B槽清洗內罩升降2馬達_軸錯誤異常
	AL403,//B槽清洗外罩升降1馬達_軸錯誤異常
	AL404,//B槽清洗外罩升降2馬達_軸錯誤異常
	AL405,//B槽噴頭擺臂升降馬達_軸錯誤異常 
	AL406,//B槽噴頭擺臂馬達_軸錯誤異常   
	AL407,//B槽頂PIN升降馬達_軸錯誤異常
	AL408,//B槽噴頭X軸馬達_軸錯誤異常   
	AL409,//B槽噴頭Y1軸馬達_軸錯誤異常  
	AL410,//B槽噴頭Y2軸馬達_軸錯誤異常  
	AL411,//B槽噴頭Z軸馬達_軸錯誤異常
	AL412,//B槽噴頭T軸馬達_軸錯誤異常 
	AL413,//B槽主軸伺服馬達_驅動器異常   
	AL414,//B槽清洗內罩升降1馬達_驅動器異常
	AL415,//B槽清洗內罩升降2馬達_驅動器異常
	AL416,//B槽清洗外罩升降1馬達_驅動器異常
	AL417,//B槽清洗外罩升降2馬達_驅動器異常
	AL418,//B槽噴頭擺臂升降馬達_驅動器異常 
	AL419,//B槽噴頭擺臂馬達_驅動器異常   
	AL420,//B槽頂PIN升降馬達_驅動器異常 
	AL421,//B槽噴頭X軸馬達_驅動器異常   
	AL422,//B槽噴頭Y1軸馬達_驅動器異常  
	AL423,//B槽噴頭Y2軸馬達_驅動器異常  
	AL424,//B槽噴頭Z軸馬達_驅動器異常   
	AL425,//B槽噴頭T軸馬達_驅動器異常   
	AL426,//                 
	AL427,//                 
	AL428,//                 
	AL429,//                 
	AL430,//清洗內罩升降1到位檢知異常    
	AL431,//清洗內罩升降2到位檢知異常    
	AL432,//清洗外罩升降1到位檢知異常    
	AL433,//清洗外罩升降2到位檢知異常    
	AL434,//噴頭X軸到位檢知異常       
	AL435,//噴頭Z軸到位檢知異常       
	AL436,//噴頭Y1軸到位檢知異常      
	AL437,//噴頭Y2軸到位檢知異常      
	AL438,//頂PIN升降到位檢知異常     
	AL439,//噴頭擺臂升降到位檢知異常     
	AL440,//噴頭擺臂擺動到位檢知異常     
	AL441,//閘門磁簧開關1(關)異常     
	AL442,//閘門磁簧開關1(開)異常     
	AL443,//閘門磁簧開關2(關)異常     
	AL444,//閘門磁簧開關2(開)異常     
	AL445,//上擺臂定位汽缸磁簧開關(定位)異常
	AL446,//上擺臂定位汽缸磁簧開關(退)異常 
	AL447,//下擺臂定位汽缸磁簧開關(定位)異常
	AL448,//下擺臂定位汽缸磁簧開關(退)異常 
	AL449,//上擺臂切換光電素子異常      
	AL450,//下擺臂切換光電素子異常      
	AL451,//DIW混CO2加熱器EGO異常  
	AL452,//DIW加熱器EGO異常      
	AL453,//漏液檢知器異常          
	AL454,//                 
	AL455,//                 
	AL456,//                 
	AL457,//                 
	AL458,//                 
	AL459,//                 
	AL460,//                 
	AL461,//                 
	AL462,//                 
	AL463,//                 
	AL464,//                 
	AL465,//                 
	AL466,//                 
	AL467,//                 
	AL468,//                 
	AL469,//                 
	AL470,//                 
	AL471,//                 
	AL472,//                 
	AL473,//                 
	AL474,//                 
	AL475,//                 
	AL476,//                 
	AL477,//                 
	AL478,//                 
	AL479,//                 
	AL480,//                 
	AL481,//                 
	AL482,//                 
	AL483,//                 
	AL484,//                 
	AL485,//                 
	AL486,//                 
	AL487,//                 
	AL488,//                 
	AL489,//                 
	AL490,//                 
	AL491,//                 
	AL492,//                 
	AL493,//                 
	AL494,//                 
	AL495,//                 
	AL496,//                 
	AL497,//                 
	AL498,//                 
	AL499,//                 
	AL500,//                 
	AL501,//                 
	AL502,//                 
	AL503,//                 
	AL504,//                 
	AL505,//                 
	AL506,//                 
	AL507,//                 
	AL508,//                 
	AL509,//                 
	AL510,//                 
	AL511,//                 
	AL512,//                 
	AL513,//                 
	AL514,//                 
	AL515,//                 
	AL516,//                 
	AL517,//                 
	AL518,//                 
	AL519,//                 
	AL520,//                 
	AL521,//                 
	AL522,//                 
	AL523,//                 
	AL524,//                 
	AL525,//                 
	AL526,//                 
	AL527,//                 
	AL528,//                 
	AL529,//                 
	AL530,//                 
	AL531,//                 
	AL532,//                 
	AL533,//                 
	AL534,//                 
	AL535,//                 
	AL536,//                 
	AL537,//                 
	AL538,//                 
	AL539,//                 
	AL540,//                 
	AL541,//                 
	AL542,//                 
	AL543,//                 
	AL544,//                 
	AL545,//                 
	AL546,//                 
	AL547,//                 
	AL548,//                 
	AL549,//                 
	AL550,//                 
	AL551,//                 
	AL552,//                 
	AL553,//                 
	AL554,//                 
	AL555,//                 
	AL556,//                 
	AL557,//                 
	AL558,//                 
	AL559,//                 
	AL560,//                 
	AL561,//                 
	AL562,//                 
	AL563,//                 
	AL564,//                 
	AL565,//                 
	AL566,//                 
	AL567,//                 
	AL568,//                 
	AL569,//                 
	AL570,//                 
	AL571,//                 
	AL572,//                 
	AL573,//                 
	AL574,//                 
	AL575,//                 
	AL576,//                 
	AL577,//                 
	AL578,//                 
	AL579,//                 
	AL580,//                 
	AL581,//                 
	AL582,//                 
	AL583,//                 
	AL584,//                 
	AL585,//                 
	AL586,//                 
	AL587,//                 
	AL588,//                 
	AL589,//                 
	AL590,//                 
	AL591,//                 
	AL592,//                 
	AL593,//                 
	AL594,//                 
	AL595,//                 
	AL596,//                 
	AL597,//                 
	AL598,//                 
	AL599 //                 
);
END_TYPE

// ---- 02_Unit/00_Alarm/E_Warn.TcDUT
{attribute 'qualified_only'}
{attribute 'strict'}
{attribute 'to_string'}
TYPE E_Warn :
(
	Warn000,
	Warn001,
	Warn002,
	Warn003,
	Warn004,
	Warn005,
	Warn006,
	Warn007,
	Warn008,
	Warn009,
	Warn010,
	Warn011,
	Warn012,
	Warn013,
	Warn014,
	Warn015,
	Warn016,
	Warn017,
	Warn018,
	Warn019,
	Warn020,
	Warn021,
	Warn022,
	Warn023,
	Warn024,
	Warn025,
	Warn026,
	Warn027,
	Warn028,
	Warn029,
	Warn030,
	Warn031,
	Warn032,
	Warn033,
	Warn034,
	Warn035,
	Warn036,
	Warn037,
	Warn038,
	Warn039,
	Warn040,
	Warn041,
	Warn042,
	Warn043,
	Warn044,
	Warn045,
	Warn046,
	Warn047,
	Warn048,
	Warn049,
	Warn050,
	Warn051,
	Warn052,
	Warn053,
	Warn054,
	Warn055,
	Warn056,
	Warn057,
	Warn058,
	Warn059,
	Warn060,
	Warn061,
	Warn062,
	Warn063,
	Warn064,
	Warn065,
	Warn066,
	Warn067,
	Warn068,
	Warn069,
	Warn070,
	Warn071,
	Warn072,
	Warn073,
	Warn074,
	Warn075,
	Warn076,
	Warn077,
	Warn078,
	Warn079,
	Warn080,
	Warn081,
	Warn082,
	Warn083,
	Warn084,
	Warn085,
	Warn086,
	Warn087,
	Warn088,
	Warn089,
	Warn090,
	Warn091,
	Warn092,
	Warn093,
	Warn094,
	Warn095,
	Warn096,
	Warn097,
	Warn098,
	Warn099,
	Warn100,
	Warn101,
	Warn102,
	Warn103,
	Warn104,
	Warn105,
	Warn106,
	Warn107,
	Warn108,
	Warn109,
	Warn110,
	Warn111,
	Warn112,
	Warn113,
	Warn114,
	Warn115,
	Warn116,
	Warn117,
	Warn118,
	Warn119,
	Warn120,
	Warn121,
	Warn122,
	Warn123,
	Warn124,
	Warn125,
	Warn126,
	Warn127,
	Warn128,
	Warn129,
	Warn130,
	Warn131,
	Warn132,
	Warn133,
	Warn134,
	Warn135,
	Warn136,
	Warn137,
	Warn138,
	Warn139,
	Warn140,
	Warn141,
	Warn142,
	Warn143,
	Warn144,
	Warn145,
	Warn146,
	Warn147,
	Warn148,
	Warn149,
	Warn150,
	Warn151,
	Warn152,
	Warn153,
	Warn154,
	Warn155,
	Warn156,
	Warn157,
	Warn158,
	Warn159,
	Warn160,
	Warn161,
	Warn162,
	Warn163,
	Warn164,
	Warn165,
	Warn166,
	Warn167,
	Warn168,
	Warn169,
	Warn170,
	Warn171,
	Warn172,
	Warn173,
	Warn174,
	Warn175,
	Warn176,
	Warn177,
	Warn178,
	Warn179,
	Warn180,
	Warn181,
	Warn182,
	Warn183,
	Warn184,
	Warn185,
	Warn186,
	Warn187,
	Warn188,
	Warn189,
	Warn190,
	Warn191,
	Warn192,
	Warn193,
	Warn194,
	Warn195,
	Warn196,
	Warn197,
	Warn198,
	Warn199,
	Warn200,
	Warn201,
	Warn202,
	Warn203,
	Warn204,
	Warn205,
	Warn206,
	Warn207,
	Warn208,
	Warn209,
	Warn210,
	Warn211,
	Warn212,
	Warn213,
	Warn214,
	Warn215,
	Warn216,
	Warn217,
	Warn218,
	Warn219,
	Warn220,
	Warn221,
	Warn222,
	Warn223,
	Warn224,
	Warn225,
	Warn226,
	Warn227,
	Warn228,
	Warn229,
	Warn230,
	Warn231,
	Warn232,
	Warn233,
	Warn234,
	Warn235,
	Warn236,
	Warn237,
	Warn238,
	Warn239,
	Warn240,
	Warn241,
	Warn242,
	Warn243,
	Warn244,
	Warn245,
	Warn246,
	Warn247,
	Warn248,
	Warn249,
	Warn250,
	Warn251,
	Warn252,
	Warn253,
	Warn254,
	Warn255,
	Warn256,
	Warn257,
	Warn258,
	Warn259,
	Warn260,
	Warn261,
	Warn262,
	Warn263,
	Warn264,
	Warn265,
	Warn266,
	Warn267,
	Warn268,
	Warn269,
	Warn270,
	Warn271,
	Warn272,
	Warn273,
	Warn274,
	Warn275,
	Warn276,
	Warn277,
	Warn278,
	Warn279,
	Warn280,
	Warn281,
	Warn282,
	Warn283,
	Warn284,
	Warn285,
	Warn286,
	Warn287,
	Warn288,
	Warn289,
	Warn290,
	Warn291,
	Warn292,
	Warn293,
	Warn294,
	Warn295,
	Warn296,
	Warn297,
	Warn298,
	Warn299,
	Warn300,
	Warn301,
	Warn302,
	Warn303,
	Warn304,
	Warn305,
	Warn306,
	Warn307,
	Warn308,
	Warn309,
	Warn310,
	Warn311,
	Warn312,
	Warn313,
	Warn314,
	Warn315,
	Warn316,
	Warn317,
	Warn318,
	Warn319,
	Warn320,
	Warn321,
	Warn322,
	Warn323,
	Warn324,
	Warn325,
	Warn326,
	Warn327,
	Warn328,
	Warn329,
	Warn330,
	Warn331,
	Warn332,
	Warn333,
	Warn334,
	Warn335,
	Warn336,
	Warn337,
	Warn338,
	Warn339,
	Warn340,
	Warn341,
	Warn342,
	Warn343,
	Warn344,
	Warn345,
	Warn346,
	Warn347,
	Warn348,
	Warn349,
	Warn350,
	Warn351,
	Warn352,
	Warn353,
	Warn354,
	Warn355,
	Warn356,
	Warn357,
	Warn358,
	Warn359,
	Warn360,
	Warn361,
	Warn362,
	Warn363,
	Warn364,
	Warn365,
	Warn366,
	Warn367,
	Warn368,
	Warn369,
	Warn370,
	Warn371,
	Warn372,
	Warn373,
	Warn374,
	Warn375,
	Warn376,
	Warn377,
	Warn378,
	Warn379,
	Warn380,
	Warn381,
	Warn382,  
	Warn383,
	Warn384,
	Warn385,
	Warn386,
	Warn387,
	Warn388,
	Warn389,  
	Warn390,
	Warn391,
	Warn392,
	Warn393,
	Warn394,
	Warn395,
	Warn396,
	Warn397,
	Warn398,
	Warn399,
	Warn400,//B槽主軸伺服馬達_驅動器異常   
	Warn401,//B槽清洗內罩升降1馬達_驅動器異常
	Warn402,//B槽清洗內罩升降2馬達_驅動器異常
	Warn403,//B槽清洗外罩升降1馬達_驅動器異常
	Warn404,//B槽清洗外罩升降2馬達_驅動器異常
	Warn405,//B槽噴頭擺臂升降馬達_驅動器異常 
	Warn406,//B槽噴頭擺臂馬達_驅動器異常   
	Warn407,//B槽頂PIN升降馬達_驅動器異常 
	Warn408,//B槽噴頭X軸馬達_驅動器異常   
	Warn409,//B槽噴頭Y1軸馬達_驅動器異常  
	Warn410,//B槽噴頭Y2軸馬達_驅動器異常  
	Warn411,//B槽噴頭Z軸馬達_驅動器異常   
	Warn412,//B槽噴頭T軸馬達_驅動器異常   
	Warn413,//
	Warn414,//
	Warn415,//
	Warn416,//
	Warn417,//
	Warn418,//
	Warn419,//
	Warn420,//
	Warn421,//
	Warn422,//
	Warn423,//
	Warn424,//
	Warn425,//
	Warn426,//
	Warn427,//
	Warn428,//
	Warn429,//
	Warn430,//
	Warn431,//
	Warn432,//
	Warn433,//
	Warn434,//
	Warn435,//
	Warn436,//
	Warn437,//
	Warn438,//
	Warn439,//
	Warn440,//
	Warn441,//
	Warn442,//
	Warn443,//
	Warn444,//
	Warn445,//
	Warn446,//
	Warn447,//
	Warn448,//
	Warn449,//
	Warn450,//
	Warn451,//
	Warn452,//
	Warn453,//
	Warn454,//
	Warn455,//
	Warn456,//
	Warn457,//                 
	Warn458,//                 
	Warn459,//                 
	Warn460,//                 
	Warn461,//                 
	Warn462,//                 
	Warn463,//                 
	Warn464,//                 
	Warn465,//                 
	Warn466,//                 
	Warn467,//                 
	Warn468,//                 
	Warn469,//                 
	Warn470,//                 
	Warn471,//                 
	Warn472,//                 
	Warn473,//                 
	Warn474,//                 
	Warn475,//                 
	Warn476,//                 
	Warn477,//                 
	Warn478,//                 
	Warn479,//                 
	Warn480,//                 
	Warn481,//                 
	Warn482,//                 
	Warn483,//                 
	Warn484,//                 
	Warn485,//                 
	Warn486,//                 
	Warn487,//                 
	Warn488,//                 
	Warn489,//                 
	Warn490,//                 
	Warn491,//                 
	Warn492,//                 
	Warn493,//                 
	Warn494,//                 
	Warn495,//                 
	Warn496,//                 
	Warn497,//                 
	Warn498,//                 
	Warn499,//                 
	Warn500,//                 
	Warn501,//                 
	Warn502,//                 
	Warn503,//                 
	Warn504,//                 
	Warn505,//                 
	Warn506,//                 
	Warn507,//                 
	Warn508,//                 
	Warn509,//                 
	Warn510,//                 
	Warn511,//                 
	Warn512,//                 
	Warn513,//                 
	Warn514,//                 
	Warn515,//                 
	Warn516,//                 
	Warn517,//                 
	Warn518,//                 
	Warn519,//                 
	Warn520,//                 
	Warn521,//                 
	Warn522,//                 
	Warn523,//                 
	Warn524,//                 
	Warn525,//                 
	Warn526,//                 
	Warn527,//                 
	Warn528,//                 
	Warn529,//                 
	Warn530,//                 
	Warn531,//                 
	Warn532,//                 
	Warn533,//                 
	Warn534,//                 
	Warn535,//                 
	Warn536,//                 
	Warn537,//                 
	Warn538,//                 
	Warn539,//                 
	Warn540,//                 
	Warn541,//                 
	Warn542,//                 
	Warn543,//                 
	Warn544,//                 
	Warn545,//                 
	Warn546,//                 
	Warn547,//                 
	Warn548,//                 
	Warn549,//                 
	Warn550,//                 
	Warn551,//                 
	Warn552,//                 
	Warn553,//                 
	Warn554,//                 
	Warn555,//                 
	Warn556,//                 
	Warn557,//                 
	Warn558,//                 
	Warn559,//                 
	Warn560,//                 
	Warn561,//                 
	Warn562,//                 
	Warn563,//                 
	Warn564,//                 
	Warn565,//                 
	Warn566,//                 
	Warn567,//                 
	Warn568,//                 
	Warn569,//                 
	Warn570,//                 
	Warn571,//                 
	Warn572,//                 
	Warn573,//                 
	Warn574,//                 
	Warn575,//                 
	Warn576,//                 
	Warn577,//                 
	Warn578,//                 
	Warn579,//                 
	Warn580,//                 
	Warn581,//                 
	Warn582,//                 
	Warn583,//                 
	Warn584,//                 
	Warn585,//                 
	Warn586,//                 
	Warn587,//                 
	Warn588,//                 
	Warn589,//                 
	Warn590,//                 
	Warn591,//                 
	Warn592,//                 
	Warn593,//                 
	Warn594,//                 
	Warn595,//                 
	Warn596,//                 
	Warn597,//                 
	Warn598,//                 
	Warn599 //                 
);
END_TYPE

// ---- 02_Unit/00_Alarm/ST_AlarmFlag.TcDUT
TYPE ST_AlarmFlag :
STRUCT
	AlarmLWord_64Bit		: ARRAY [0..2] OF LWORD;
	WarningLWord_64Bit		: ARRAY [0..1] OF LWORD;
END_STRUCT
END_TYPE

// ---- 02_Unit/00_Alarm/ST_AlarmItem.TcDUT
TYPE ST_AlarmItem :
STRUCT
	Reset					: BOOL;		//異常復歸輸出
	R_Trig_AlarmReset		: R_TRIG;	//異常復歸上微分
	F_Trig_Error			: F_TRIG;	//異常發生下微分
	Error					: BOOL;		//錯誤發生
	Warning					: BOOL;		//警示發生
	Alarm					: BOOL;		//異常發生
	Rescue					: BOOL;		//過溫救貨中 (AlarmList[12..15] 任一觸發且無其他 alarm)
	ErrorCounts				: INT;		//錯誤數量
	WarningCounts			: INT;		//警示數量
	AlarmCounts				: INT;		//異常數量      
END_STRUCT
END_TYPE

// ---- 02_Unit/00_Alarm/U_Alarm.TcDUT
TYPE U_Alarm :
UNION
	Item			:ST_AlarmParameter;
	Row				:ARRAY[0..599] OF INT;
END_UNION
END_TYPE

// ---- 02_Unit/01_Customization/ST_Parameter.TcDUT
TYPE ST_Parameter :
STRUCT
	strName						:STRING(50);
	//拆箱 
	Unboxing_PullOut			:REAL;			//出紙箱位置 
	Unboxing_LoadOut			:REAL;			//推出位置 
	Unboxing_Velo				:REAL;			//運行速度 
	Unboxing_DelayTime			:ARRAY [0..2] OF TIME;			
	
	
	//雙伺服環形參數 
	Dual_LoadInQty				:ARRAY [0..9]	OF INT;	//每層數量
	Dual_LoadInPos				:REAL;			//環形接料點
	Dual_LoadOutPos				:REAL;			//環形出料點_RB 
	Dual_LoadOutSecPos			:REAL;			//環形出料2點_RB 
	Dual_ModuleSlotQty			:UINT;			//輸送帶格數 
	Dual_ModulePitchLength		:REAL;			//每格長度
	Dual_Length					:REAL;			//輸送帶長
	Dual_Velo					:REAL;			//運行速度 
	Dual_Gap					:REAL;			//安全間距
	Dual_TwiceClip				:BOOL;			//兩次夾取  
	
	//入料輸送
	Fly_Disdance				:REAL;		//輸送帶偵測料件輸送距離 
	Fly_Velo					:REAL;
	Fly_DelayTime				:TIME;
	
	//裝箱參數 
	Load_Sdandby			:REAL;			//預備位置 
	Load_RBLoadin			:REAL;			//手臂入料位置
	Load_LoadOut			:REAL;			//推出位置 	
	Load_Velo				:REAL;			//速度
	Load_RBPrgNo			:BYTE;
	Load_Type			:UINT;				//1= 四夾 , 2= 兩夾
	Load_RBVelo			:BYTE;
	//產品資訊  
	PackagingPicQuantity		:INT;		//每箱包裝數量   
	PackagingBoxQuantity		:INT;		//盒棧箱數量 
	PackagingWeight			:REAL;			//包裝重量 
	PackagingWeightUpLimit	:REAL;
	PackagingWeightLowLimit	:REAL;				
	PackagingCheck			:BOOL;
	PackagingBarcode		:BOOL;
	PackagingHaltAuto		:BOOL;
	
	//震動 
	shock_HighTime				:TIME;
	shock_DelayTime				:TIME;
	//推疊 
	stack_bUsed					:BOOL;
	stack_DelayTime1			:TIME;
	stack_DelayTime2			:TIME;
	//堆棧  
	StackingRB_DelayTime1			:TIME;
	StackingRB_DelayTime2			:TIME;	
	StackingRB_LayerData			:ARRAY [0..2]	OF INT;;
	StackingRB_RBPrgNo				:BYTE;
	StackingRB_length					:INT;
	StackingRB_width					:INT;
	StackingRB_height					:INT;
	StackingRB_RBVelo			:BYTE;
	
	
END_STRUCT
END_TYPE

// ---- 02_Unit/01_Customization/ST_SlotData.TcDUT
TYPE ST_SlotData :
STRUCT
	ScanIn:BOOL;
	LoadIn:BOOL;
	LatchPosition :LREAL;
	GearInPosition:LREAL;
END_STRUCT
END_TYPE

// ---- 02_Unit/02_Cylinder kit/E_CylFault.TcTLEO
{attribute 'strict'}
{attribute 'qualified_only'}
{attribute 'to_string'}
TYPE E_CylFault :
(
	None                  := 0,
    TimeoutExtend         := 1,  // 預期伸出但到位逾時
    TimeoutRetract        := 2,  // 預期縮回但到位逾時
    BothSensorsOn         := 3,  // 原點與末端同時為真（邏輯矛盾/配線錯）
    CoilConflict          := 4,  // 兩線圈同時為真（監測到）
    SensorStuck           := 5   // 感測卡住（可選，見下方邏輯）
);
END_TYPE

// ---- 02_Unit/02_Cylinder kit/E_CylinderType.TcTLEO
{attribute 'strict'}
{attribute 'to_string'}
TYPE E_CylinderType :
(
    ThreePort_TwoPosition := 0,   // 3口2位
    FivePort_TwoPosition  := 1    // 5口2位
);
END_TYPE

// ---- 02_Unit/02_Cylinder kit/ST_Cylinder.TcDUT
TYPE ST_Cylinder :
STRUCT
    // --- 硬體輸出 ---
    qExtendCoil        AT %Q* : BOOL;  // 氣缸伸出線圈
    qRetractCoil       AT %Q* : BOOL;  // 氣缸收回線圈

    // --- 硬體輸入 ---
    iOriginSensor      AT %I* : BOOL;  // 原點感測
    iEndSensor         AT %I* : BOOL;  // 末端感測

    // --- 軟體旗標 ---
    bOriginConfirmed        : BOOL;  // 原點信號已確認（延時/除抖後）
    bEndConfirmed           : BOOL;  // 末端信號已確認（延時/除抖後）
    bError                  : BOOL;  // 通用錯誤旗標
	bReset					: BOOL;
	eCylFault				: E_CylFault; //異常狀態
	
	// --- 名稱 ---	{attribute 'TcEncoding':='UTF-8'}
	strName					: WSTRING(32);
	// --- 參數 ---
	stCylinderPara     		: ST_CylinderParameter;  
	
END_STRUCT
END_TYPE

// ---- 02_Unit/02_Cylinder kit/ST_CylinderParameter.TcDUT
TYPE ST_CylinderParameter :
STRUCT
    eCylinderType      : E_CylinderType;  // 氣缸型式 (3/2 或 5/2)
    // --- 末端 (End) 相關 ---
    bEndNoSensor       : BOOL;            // 末端無感測模式
    tEndDebounceTime   : TIME;            // 末端除抖/穩定判定時間
    tEndTimeout        : TIME;            // 末端動作超時
    // --- 原點 (Origin) 相關 ---
    bOriginNoSensor    : BOOL;            // 原點無感測模式
    tOriginDebounceTime: TIME;            // 原點除抖/穩定判定時間
    tOriginTimeout     : TIME;            // 原點動作超時
    // --- 共用 ---
    bCoilAutoOff       : BOOL;            // 動作完成自動斷電
END_STRUCT
END_TYPE

// ---- 02_Unit/11_EventLogger/E_EventType.TcTLEO
{attribute 'qualified_only'}
{attribute 'strict'}
{attribute 'to_string'}
TYPE E_EventType :
(
    Verbose  := 0, 
    Info     := 1, 
    Warning  := 2, 
    Error    := 3, 
    Critical := 4
);
END_TYPE

// ---- 02_Unit/11_EventLogger/ST_Event.TcDUT
TYPE ST_Event :
STRUCT
	eEventType		: E_eventType ;	// Verbose:= 0, Info := 1, Warning  := 2,  Error := 3, Critical := 4
	nEventIdentity	: UDINT ;
	strEventText	: STRING(50);
	dtTimeStamp		: DATE_AND_TIME;
END_STRUCT
END_TYPE

// ---- 02_Unit/99_Other/ST_Operation.TcDUT
TYPE ST_Operation :
STRUCT
	bInitialSign		:BOOL;	//初始化驅動 
	xInitialDone		:BOOL;	//初始化完成 
	xInitialRuning		:BOOL;	//初始化運行中 
	bChangeMode			:BOOL;	//切換PLC狀態 
	xAutoMode			:BOOL;	//自動狀態 
	bStop_Sign			:BOOL;	//停止訊號  
	xAutoRuning			:BOOL;	//自動運行中 
	bCycleStep			:BOOL;	//半自動 
	bStart				:BOOL;
	strStatusText		:WSTRING(100);
	bReset				:BOOL;	//RESET
END_STRUCT
END_TYPE

// ---- 00_GVLs/HardwareIO.TcGVL
VAR_GLOBAL
	(*EtherCAT Link Status*)
	MainFiledBus		AT%I*		:ARRAY [0..20] OF UINT;
	
	
	
	(*DO*)	
	EL2889	AT%Q*	:ARRAY [1..3,1..16]OF BOOL;
	(*DI*)
	EL1889	AT%I*	:ARRAY [1..4,1..16]OF BOOL;
	(*RB*)
	RB_CS				:RB_KR_PickPlace;
	RB_CS_SysIO			:ST_CS_sysIO;
	RB_CS_PickIO		:ST_CS_PickIO;

	RB_KR_SysIO			:ST_KR_sysIO := (qDRIVES_OFF := TRUE, qMOVE_ENABLE := TRUE);	
	RB_KR_StackingIO	:ST_KR_stackingIO;
	RB_KR				:RB_KR_Stacking;

	(*伺服馬達 *)
	Axis_DualServo1	 						:AXIS_REF_EXT;	//雙伺服-左 
	Axis_DualServo2							:AXIS_REF_EXT;	//雙伺服-右	
	Axis_FlyIn								:AXIS_REF_EXT;	//入料輸送-飛入 
	Axis_BoxPullOut							:AXIS_REF_EXT;	//拉紙箱伺服 
	Axis_load1								:AXIS_REF_EXT;	//推出紙箱-右 
	Axis_load2								:AXIS_REF_EXT;	//推出紙箱-左  
	
	(*一般傳動 *)
	Motor_LoadIn							:ST_Inventer;	//入口托速馬達  
	Motor_Blower							:ST_Inventer;	//鼓風機 
	Motor_LoadPurge1,Motor_LoadPurge2		:ST_Inventer;	//入口排放馬達    
 
	Roller_Purge							:ST_Inventer;	//排出滾輪  
	Roller_Exit								:ST_Inventer;	//出口滾輪 
	
	//紙箱入料 
	Cyl_BoxSidePitch						:ST_Cylinder := (stCylinderPara := (tEndTimeout := TIME#1s0ms, tOriginTimeout := TIME#1s0ms));
	Cyl_BoxSideBottom						:ST_Cylinder := (stCylinderPara := (tEndTimeout := TIME#1s0ms, tOriginTimeout := TIME#1s0ms));
	Sen_BoxsideFeed							AT%I*	:BOOL;
	Sen_BoxsideStorageMaterial				AT%I*	:BOOL;
	//取紙箱馬達  
	Cyl_AxisBoxCatch						:ST_Cylinder := (stCylinderPara := (tEndTimeout := TIME#3S0MS, tOriginTimeout := TIME#5S0MS));	//取箱汽缸 
	Sen_AxisBoxCatchVacumm			AT%I*	:BOOL;
	Vacm_AxisCatchBox				AT%Q*	:BOOL;
	Sen_AxisBoxORG					AT%I*	:BOOL;
	Cyl_Axis90								:ST_Cylinder := (stCylinderPara := (tEndTimeout := TIME#1S0MS, tOriginTimeout := TIME#1S0MS));	//90度 
	Sen_Axis90Vacumm				AT%I*	:BOOL;
	Vacm_Axis90						AT%Q*	:BOOL;
	Cyl_AxisBottom							:ST_Cylinder := (stCylinderPara := (tEndTimeout := TIME#1S0MS, tOriginTimeout := TIME#1S0MS));	//底部壓和 
	
	//封箱底 
	Motor_BoxSealBottom_L					:ST_Inventer;	//封箱底馬達-L 
	Motor_BoxSealBottom_R					:ST_Inventer;	//封箱底馬達-R 
	Cyl_BeltBottom							:ST_Cylinder := (stCylinderPara := (tEndTimeout := TIME#1S0MS, tOriginTimeout := TIME#1S0MS));	//皮帶底部壓和 
	Cyl_BeltBottomSup						:ST_Cylinder;	//皮帶底部壓和邊角 沒感測器  
	Sen_BeltLoadIn					AT%I*	:BOOL;	
	Sen_BeltLoadOut					AT%I*	:BOOL;
	//UNLOAD紙箱區域  
	Cyl_UnloadDef						:ST_Cylinder := (stCylinderPara := (tEndTimeout := TIME#2s0ms, tOriginTimeout := TIME#2s0ms));	//上方定型汽缸
	Sen_UnloadLoadIn					AT%I*	:BOOL;
	Sen_UnloadLoadPos					AT%I*	:BOOL;
	Sen_AxisLoad1ORG					AT%I*	:BOOL;
	Sen_AxisLoad2ORG					AT%I*	:BOOL;

	//轉彎區域 NG 
	Sen_TFLoadIn					AT%I*	:BOOL;
	Sen_NGLoadOut					AT%I*	:BOOL;
	Roller_LoadcellIn						:ST_Inventer;	//滾輪秤重進入  
	Roller_LoadcellOut						:ST_Inventer;	//滾輪秤重橫向皮帶  
	Roller_LoadcellUD						:ST_InventerUD;	//滾輪秤重航向頂上	
	AssRoller								:FB_RollRightAngle;
	
	
	Cyl_NGPurge							:ST_Cylinder:= (stCylinderPara := (tEndTimeout := TIME#1s0ms, bOriginNoSensor := TRUE, tOriginDebounceTime := TIME#500ms));	//NG推出汽缸   
	Swtich_PassFeet						AT%I*	:BOOL;
	Cyl_ShockStop							:ST_Cylinder := (stCylinderPara := (bEndNoSensor := TRUE, tEndDebounceTime := TIME#500ms, tOriginTimeout := TIME#1s0ms));	//震動出口stooper   
	Sen_ShockPos						AT%I*	:BOOL;
	Motor_shock								:ST_Inventer;	//震動馬達 
	
	//疊箱 
	Cyl_StackUD								:ST_Cylinder := (stCylinderPara := (tEndTimeout := TIME#2s0ms, tOriginTimeout := TIME#2s0ms));	//疊箱  
	Sen_StackUDVacumm				AT%I*	:BOOL;
	Sen_StackComvStop				AT%I*	:BOOL;
	Vacm_StackUD					AT%Q*	:BOOL;
	Motor_Stack								:ST_Inventer;	//疊箱馬達
	
	//出口區域 
	Sen_ExitLoadIn				AT%I*	:BOOL;	
	Sen_ExitComvStop			AT%I*	:BOOL;	
	Sen_ExitBoxCheck			AT%I*	:BOOL;	
	Cyl_ExitClip						:ST_Cylinder;
	Cyl_ExitStopper						:ST_Cylinder;
	
	//高速入料 
	Cyl_FlyIn_Pass				AT%Q*		:BOOL;
	
	//捆包機 
	Bundling_ErrorSignal			AT%I*	:BOOL;	
	Bundling_yPause					AT%Q*	:BOOL;	

	(*其他 *)
	PB_Start			AT%I*	:BOOL;
	PB_Stop				AT%I*	:BOOL;
	PB_EMG				AT%I*	:BOOL;
	Light_Green			AT%Q*	:BOOL;
	Light_Red			AT%Q*	:BOOL;
	Light_Yellow			AT%Q*	:BOOL;
	Light_BZ			AT%Q*	:BOOL;
	ElectronicBoxLight	AT%Q*	:BOOL;
	WindowsSafe			AT%I*	:ARRAY [1..6] OF BOOL;			//4=Gate 5btn
	Air_Signal			AT%I*	:BOOL;	
	TemperatureHigh			AT%I*	:BOOL;	
	TemperatureFans			AT%Q*	:BOOL;
	
	LoadCell		:FB_EL3356_0010;//秤重單元 
END_VAR

// ---- 00_GVLs/Parameter_PERSISTENT.TcGVL
VAR_GLOBAL PERSISTENT 
	//Parameter	:ST_Parameter := (ConveyorVelo:=300,RollerVelo:= 300,Roll_LoadInPos := 1300, Roll_LoadOutPos := 2200, Roll_ConveyorLength := 3520, Roll_ModuleSlotQty := 4, Roll_ModuleLength := 150, ConvGap := 50, ConveyorTrasnfeDisdance:= 300)	;
	//ORG Offset
	Setting_Dual1_ORG_Offset	:REAL;
	Setting_Dual2_ORG_Offset	:REAL;
	Setting_Dual2_ORG_Velo		:REAL;
	Setting_DualServoAcc		:REAL;
	Setting_DualServoDec		:REAL;
	Setting_DualServoJerk		:REAL;

	Setting_Unload1_ORG_Offset	:REAL;
	Setting_Unload2_ORG_Offset	:REAL;
	Setting_Unload2_ORG_Velo	:REAL;	
	Setting_Dual_ConveyorLength			:REAL;			//雙伺服輸送帶總長 3657.5
	Setting_Load_ConveyorLength			:REAL;			//裝箱輸送帶總長 
	
	Setting_FanAuto					:BOOL;			//風扇自動 
	Setting_DualServoCalibration	:BOOL;			//雙伺服輸送校準 
	///////////////////////////////////////////////////	
	EventLogger 				: EventLogger;
	RunParameter				:ST_Parameter 	;
	//////////////////Loadcell/////////////////////////////////
	Setting_MaxLoad			:REAL;
	Setting_RefLoad			:REAL;
	Setting_LoadPercent		:REAL;
	///////////////////////////////
	Counter_Pallet			:WORD;	//已完成棧板
	Counter_ExitBox			:WORD;	//已出箱 
	Counter_PackLoadIn		:DWORD;	//已入包裝 
	Counter_OKBox			:WORD;	//完成裝箱 
	Counter_NGBox			:WORD;	//NG裝箱 
	
END_VAR

// ---- 00_GVLs/GVL.TcGVL
VAR_GLOBAL
	OP		:ST_Operation	;
	SF		:Spacil_FC;
	slot	:ARRAY [1..5] OF ST_SlotData;
	DualGroupRef 		: AXES_GROUP_REF;
	M_Openbox1			:Ass_Openbox;				// 
	M_DualServo			:Ass_DualServo;				//雙伺服輸送
	M_LoadPic3			:Ass_LoadPic;				//裝箱 
	M_Sealing2			:Ass_Sealing;				//封箱底部 
	M_UnloadNG4			:Ass_UnloadNG;				//
	M_StackComv5		:Ass_StackComv;				//推疊機構 
	M_RBStack6			:Ass_RBStack;				//手臂堆疊 
	M_Pallet			:Ass_Pallet;
	RecipeManCommands	:RecipeManCommands;			//配方處理 
	MainControl			:MainControl;
	DoNotLoadingRB: BOOL;
END_VAR

// ---- 00_GVLs/HMI_Mapp.TcGVL
VAR_GLOBAL
	Edit_Parameter	:ST_Parameter 	;
	Hmi_bDualAutoTest		:BOOL;
	Hmi_bDualFeedTest		:BOOL;
	Hmi_bDualAutoTestTime	:TIME;
	
	Hmi_bPickAutoTest		:BOOL;
	Hmi_bPickAutoTestTime	:TIME;
	Hmi_bPickFeedTest		:BOOL;
	
	Hmi_bBoxAutoTest		:BOOL;
	Hmi_bBoxAutoTestTime	:TIME;
	Hmi_bBoxFeedTest		:BOOL;		
	//換詹版
	Hmi_bAutoChangePallet	:BOOL;
	Hmi_bChangePalletbtn	:BOOL;
	Hmi_bChangePalletDemand	:BOOL;
END_VAR

// ---- 02_Unit/01_Customization/ITF_AutoStructCommand.TcIO
INTERFACE ITF_AutoStructCommand

PROPERTY Connect : String(50)
GET
END_GET
SET
END_SET
END_PROPERTY

PROPERTY Error : BOOL
GET
END_GET
END_PROPERTY

METHOD ErrorClear : BOOL
VAR_INPUT
END_VAR
END_METHOD

METHOD FB_init : BOOL
VAR_INPUT
	bInitRetains : BOOL; // if TRUE, the retain variables are initialized (warm start / cold start)
	bInCopyCode : BOOL;  // if TRUE, the instance afterwards gets moved into the copy code (online change)
END_VAR
END_METHOD

METHOD HaltStepContiune : BOOL
VAR_INPUT
END_VAR
END_METHOD

METHOD Initialization : BOOL
VAR_INPUT
	_Testmode	:BOOL;
END_VAR
END_METHOD

PROPERTY NoEntry : BOOL	//不允許進入
GET
END_GET
END_PROPERTY

METHOD Pause : BOOL
VAR_INPUT
END_VAR
END_METHOD

METHOD Process : BOOL
VAR_INPUT
	bHlatMode	:BOOL;
END_VAR
END_METHOD

PROPERTY Status : STRING(50)
GET
END_GET
END_PROPERTY

END_INTERFACE

// ---- 01_POUs/static/Recipe_POU.TcPOU
PROGRAM Recipe_POU
VAR	
	bLoadDefData		:BOOL;
	bCreateRecipe		:BOOL;
	bSaveParameter 		:BOOL;  //保存文件 
	bLoadParameter 		:BOOL;  //讀取文件 
	bDelete				:BOOL;	//刪除配方 
	bRecipeCount		:BOOL	:=TRUE;	//讀取配方數量
	bSaveView,bLoadView,bCreateView		:BOOL;
	dwError				:DWORD;
	sRecipeName			:STRING(50);
    arrFileName : ARRAY[1..100] OF STRING;
	arrFileBtn 	: ARRAY[1..100] OF BOOL;
	bCopytoWork	:BOOL;
	i,RecipeQty: INT;
	bTest,bPreview: BOOL;
END_VAR

VAR CONSTANT
	//參數數量
	QuantityLimit	:INT := 100;
END_VAR

FOR i:= 1 TO QuantityLimit DO
	IF arrFileBtn[i] THEN
		Edit_Parameter.strName	:= arrFileName[i];
		RunParameter.strName	:= arrFileName[i];
		arrFileBtn[i]:=FALSE;
	END_IF
END_FOR
Edit_Parameter.strName:= F_TrimRightSpace(Edit_Parameter.strName);
sRecipeName	:= Edit_Parameter.strName;

/////////////讀取recipeQty /////////////////
IF bRecipeCount THEN
	ReloadList();
	bRecipeCount:=FALSE;
END_IF;
//将plc数据以文件形式保存在工控机中 

CheckCreateView();
IF bCreateRecipe THEN
	dwError	:=RecipeManCommands.CreateRecipe(RecipeDefinitionName:='Recipes' , RecipeName:=sRecipeName );
	dwError	:=RecipeManCommands.ReadAndSaveRecipe(RecipeDefinitionName:='Recipes' , RecipeName:=sRecipeName );
	ReloadList();
	bCreateRecipe :=FALSE;
END_IF
//将工控机中的文件数据读取到plc中 
CheckLoadView();
IF bLoadParameter THEN
	dwError	:=	0;
    dwError:= RecipeManCommands.LoadAndWriteRecipe(RecipeDefinitionName:='Recipes' , RecipeName:=sRecipeName);
    bLoadParameter:=FALSE;
END_IF 
IF bSaveParameter THEN  
	dwError	:=RecipeManCommands.ReadAndSaveRecipe(RecipeDefinitionName:='Recipes' , RecipeName:=sRecipeName );
	bSaveParameter:=FALSE;
END_IF

IF bTest THEN
	dwError	:=RecipeManCommands.ReloadRecipes(RecipeDefinitionName:='Recipes' );
	bTest:=FALSE;
END_IF

IF bDelete THEN
	dwError	:=RecipeManCommands.DeleteRecipe(RecipeDefinitionName:='Recipes' , RecipeName:=sRecipeName );
	dwError	:=RecipeManCommands.DeleteRecipeFile(RecipeDefinitionName:='Recipes' , RecipeName:=sRecipeName );
	ReloadList();
	bDelete	:=FALSE;
END_IF
IF bCopytoWork THEN
	bCopytoWork:=FALSE;
	RunParameter:= Edit_Parameter;
END_IF

IF bPreview THEN
	RunParameter.strName:= F_TrimRightSpace(RunParameter.strName);
	dwError:= RecipeManCommands.LoadAndWriteRecipe(RecipeDefinitionName:='Recipes' , RecipeName:=RunParameter.strName);	
	bPreview:= FALSE;
	IF dwError<> 0 THEN
		EventLogger.eEventType		:= 2;
		EventLogger.strEventText	:= 'Recipe Not Find ';	
		EventLogger();
		ELSE	
		RunParameter	:= Edit_Parameter;
		EventLogger.eEventType		:= 1;
		EventLogger.strEventText	:= 'Recipe Loaded ';	
		EventLogger();
	END_IF
END_IF

IF bLoadDefData THEN
	LoadDefData();
	bLoadDefData:=FALSE;
END_IF

ACTION CheckCreateView:
IF sRecipeName='' THEN
	bCreateView:=FALSE;
	RETURN;
END_IF
//確認數量不超過 
IF RecipeQty < QuantityLimit THEN
	bSaveView	:=FALSE;
	bLoadView	:=FALSE;
	bCreateView:=TRUE;
END_IF

FOR i := 1 TO QuantityLimit DO
	IF sRecipeName = arrFileName[i] THEN
		bCreateView:=FALSE;
		EXIT;
	END_IF
END_FOR
END_ACTION

ACTION CheckLoadView:
bLoadview:=FALSE;
bSaveView:=FALSE;
IF sRecipeName='' THEN
	RETURN;
END_IF

FOR i := 1 TO QuantityLimit DO
	IF sRecipeName = arrFileName[i] THEN
		bLoadview:= bSaveView:=TRUE;
		EXIT;
	END_IF
END_FOR
IF Edit_Parameter.Dual_Velo = 0 OR Edit_Parameter.Fly_Velo = 0 THEN
	bSaveView:=FALSE;
END_IF
END_ACTION

ACTION LoadDefData:
Edit_Parameter.Dual_LoadInPos			:= 1500;
Edit_Parameter.Dual_ModulePitchLength	:= 100;
Edit_Parameter.Dual_Length				:= 430;
Edit_Parameter.Dual_Gap					:= 150;
Edit_Parameter.Dual_LoadOutPos			:= 2800;
Edit_Parameter.Dual_LoadOutSecPos		:= 3200;
Edit_Parameter.Dual_TwiceClip			:= FALSE;
Edit_Parameter.Dual_Velo				:= 1000;
Edit_Parameter.Dual_LoadInQty[0]		:= 4;
Edit_Parameter.Dual_LoadInQty[1]		:= 4;
Edit_Parameter.Dual_LoadInQty[2]		:= 4;
Edit_Parameter.Dual_LoadInQty[3]		:= 4;


Edit_Parameter.Fly_DelayTime			:= T#0.2S;
Edit_Parameter.Fly_Disdance				:= 700;
Edit_Parameter.Fly_Velo					:= 1000;

Edit_Parameter.Unboxing_PullOut			:= 320;
Edit_Parameter.Unboxing_LoadOut			:= 525;
Edit_Parameter.Unboxing_Velo			:= 150;

Edit_Parameter.Load_Sdandby				:= 0;
Edit_Parameter.Load_RBLoadin			:= 300;
Edit_Parameter.Load_Velo				:= 200;
Edit_Parameter.Load_LoadOut				:= 0;		//暫無使用
END_ACTION

METHOD LoadingRecipe : BOOL
VAR_INPUT
	Name			:STRING(50);
END_VAR

VAR
	bGetRecipe: BOOL;
END_VAR
IF Name='' THEN
	LoadingRecipe:=FALSE;
	RETURN;
END_IF
bGetRecipe:=FALSE;
FOR i := 1 TO QuantityLimit DO
	IF Name = arrFileName[i] THEN
		bGetRecipe:=TRUE;
		EXIT;
	END_IF
END_FOR
END_METHOD

ACTION ReloadList:
	FOR i :=1 TO QuantityLimit DO
		arrFileName[i] := '';
	END_FOR
	
	dwError := RecipeManCommands.ReloadRecipes('Recipes');
	RecipeQty:= RecipeMancommands.GetRecipeCount('Recipes');
	IF dwError = 0 THEN
		dwError := RecipeManCommands.GetRecipeNames(
		RecipeDefinitionName := 'Recipes',
		pStrings := ADR(arrFileName),
		iSize := 50,
		iStartIndex := 0);
	END_IF
END_ACTION

END_PROGRAM

// ---- 02_Unit/99_Other/F_TrimRightSpace.TcPOU
FUNCTION F_TrimRightSpace : STRING
VAR_INPUT
	 strIn : STRING;
END_VAR
VAR
	  nLen : INT;
END_VAR

F_TrimRightSpace := strIn;

	nLen := LEN(F_TrimRightSpace);
	
	WHILE (nLen > 0) AND MID(F_TrimRightSpace,1,nLen)=' ' DO
		nLen := nLen - 1;
	END_WHILE
	F_TrimRightSpace := LEFT(F_TrimRightSpace, nLen);

END_FUNCTION

// ---- 02_Unit/11_EventLogger/EventLogger.TcPOU
FUNCTION_BLOCK PUBLIC EventLogger
VAR_INPUT
	eEventType : E_eventType ;
	nEventIdentity : UDINT ;
	strEventText	: STRING(255);
END_VAR

VAR
	EventBuffer : ARRAY [1..Max_Size_OF_Buffer] OF ST_Event;
	CurrentEventBufferIndex : INT:= 0;
	i 						: INT;
END_VAR

VAR CONSTANT
	Max_Size_OF_Buffer : INT := 100;
END_VAR

FOR i :=  Max_Size_OF_Buffer TO 2 BY -1 DO 
	EventBuffer[i]:= EventBuffer[i-1];
END_FOR
EventBuffer[1].eEventType := eEventType;
EventBuffer[1].nEventIdentity	:= nEventIdentity;
EventBuffer[1].strEventText	:= strEventText;
UpdateEventTimeWithSystemTime(stEvent := EventBuffer[1]);

END_FUNCTION_BLOCK

// ---- 02_Unit/11_EventLogger/UpdateEventTimeWithSystemTime.TcPOU
FUNCTION UpdateEventTimeWithSystemTime  
VAR_INPUT
	stEvent :REFERENCE TO ST_Event;
END_VAR
	
VAR
	fbLocalSystemTime	:FB_LocalSystemTime := (bEnable := TRUE);
	fbGETSYSTEMTIME 	:GETSYSTEMTIME;
	stT_FILETIME		:T_FILETIME;
END_VAR



stEvent.dtTimeStamp:= SF.systemTime;

END_FUNCTION

// ---- 01_POUs/static/prgInputMapp.TcPOU
PROGRAM prgInputMapp
VAR
END_VAR

;

END_PROGRAM

// ---- 01_POUs/static/Device_POU.TcPOU
PROGRAM Device_POU
VAR
	fbCylinderBase:ARRAY [0..20] OF  FB_CylinderBase;
END_VAR


// PAGE Axis_Conf
Axis_DualServo1(EMG := Not PB_EMG, Enable_Positive := TRUE); // AXIS_REF_Ext
Axis_FlyIn(EMG := Not PB_EMG, Enable_Positive := TRUE); // AXIS_REF_Ext
Axis_DualServo2(EMG := Not PB_EMG, Enable_Positive := TRUE); // AXIS_REF_Ext
Axis_BoxPullOut(EMG := Not PB_EMG, Enable_Positive := TRUE, Enable_Negative := TRUE); // AXIS_REF_Ext
Axis_load1(EMG := Not PB_EMG, Enable_Positive := TRUE); // AXIS_REF_Ext
Axis_load2(EMG := Not PB_EMG, Enable_Positive := TRUE); // AXIS_REF_Ext

// PAGE Cylinder_Conf
fbCylinderBase[1](i_en := TRUE, ref_stCyl := Cyl_AxisBoxCatch); // FB_CylinderBase
fbCylinderBase[0](i_en := TRUE, ref_stCyl := Cyl_BoxSideBottom); // FB_CylinderBase
fbCylinderBase[2](i_en := TRUE, ref_stCyl := Cyl_Axis90); // FB_CylinderBase
fbCylinderBase[4](i_en := TRUE, ref_stCyl := Cyl_UnloadDef); // FB_CylinderBase
fbCylinderBase[3](i_en := TRUE, ref_stCyl := Cyl_AxisBottom); // FB_CylinderBase

// PAGE Assamble
M_StackComv5(); // Ass_StackComv
M_Sealing2(); // Ass_Sealing
M_UnloadNG4(); // Ass_UnloadNG
M_DualServo(); // Ass_DualServo
M_Openbox1(); // Ass_Openbox
M_LoadPic3(); // Ass_LoadPic
M_RBStack6(); // Ass_RBStack
AssRoller(ref_Roller := Roller_LoadcellIn, ref_Belt := Roller_LoadcellOut, ref_UD := Roller_LoadcellUD); // FB_RollRightAngle

// PAGE Other
LoadCell(); // FB_EL3356_0010
RB_CS(); // RB_KR_PickPlace
RB_KR(); // RB_KR_Stacking
SF(); // Spacil_FC
MainControl();

END_PROGRAM

// ---- 02_Unit/02_Cylinder kit/FB_CylinderBase.TcPOU
FUNCTION_BLOCK FB_CylinderBase 
VAR_INPUT
	i_en					:BOOL;
	ref_stCyl              : REFERENCE TO ST_Cylinder;  // 綁定目標 
END_VAR
VAR
    // 既有：除抖與監看 
	_tonTimeOutEnd,_tonEndDeb		:TON;	
	_tonTimeOutORI,_tonORIDeb		:TON;
    // === ConsistencyCheck 專用的「保留狀態」 === 
    _cc_tonStuck   : TON;   // 感測卡住用；放在 FB 內才能跨掃描記憶 
	
	
END_VAR

IF NOT i_en THEN
	RETURN;
END_IF

// === 確認使用的型號 ===  
CASE ref_stCyl.stCylinderPara.eCylinderType OF 
	E_CylinderType.ThreePort_TwoPosition:
		ThreePort_TwoPosition();
	E_CylinderType.FivePort_TwoPosition:
		FivePort_TwoPosition();
END_CASE

_cc_tonStuck(IN:= ref_stCyl.iEndSensor AND ref_stCyl.iOriginSensor , PT:=T#0.3S);
IF _cc_tonStuck.Q THEN
	ref_stCyl.eCylFault	:= E_CylFault.BothSensorsOn;
END_IF
IF ref_stCyl.bReset THEN
	ref_stCyl.bReset:=FALSE;
	Reset();
END_IF


_UpdateFaultFlag();

METHOD PRIVATE _UpdateFaultFlag : BOOL
VAR_INPUT
END_VAR
ref_stCyl.bError := (ref_stCyl.eCylFault <> E_CylFault.None) ;
END_METHOD

METHOD INTERNAL FivePort_TwoPosition
VAR_INPUT
END_VAR
//異常感測時間	
	_tonTimeOutEnd(IN := ref_stCyl.qExtendCoil AND NOT ref_stCyl.iEndSensor, PT := ref_stCyl.stCylinderPara.tEndTimeout);
	
	IF _tonTimeOutEnd.Q AND NOT ref_stCyl.stCylinderPara.bEndNoSensor THEN		//確認TimeOut + NO Sensor 
		ref_stCyl.eCylFault := E_CylFault.TimeoutExtend;
	END_IF

	_tonTimeOutORI(IN := ref_stCyl.qRetractCoil AND NOT ref_stCyl.iOriginSensor, PT := ref_stCyl.stCylinderPara.tOriginTimeout);
	
	IF _tonTimeOutORI.Q AND NOT ref_stCyl.stCylinderPara.bOriginNoSensor THEN		//確認TimeOut + NO Sensor 
		ref_stCyl.eCylFault := E_CylFault.TimeoutRetract;
	END_IF	

	
//穩定時間 輸出監控 
	
	IF NOT ref_stCyl.stCylinderPara.bEndNoSensor  THEN			//有感測器 
		_tonEndDeb(IN:=ref_stCyl.iEndSensor , PT := ref_stCyl.stCylinderPara.tEndDebounceTime );
		ref_stCyl.bEndConfirmed	:= _tonEndDeb.Q ;
	ELSE														//沒感測器 
		_tonEndDeb(IN:=ref_stCyl.qExtendCoil , PT := ref_stCyl.stCylinderPara.tEndDebounceTime );
		ref_stCyl.bEndConfirmed	:= _tonEndDeb.Q ;		
	END_IF

	
//穩定時間 回歸

	IF NOT ref_stCyl.stCylinderPara.bOriginNoSensor  THEN			//有感測器 
		_tonORIDeb(IN:=ref_stCyl.iOriginSensor , PT := ref_stCyl.stCylinderPara.tOriginDebounceTime );
		ref_stCyl.bOriginConfirmed	:= _tonORIDeb.Q ;
	ELSE														//沒感測器  
		_tonORIDeb(IN:= ref_stCyl.qRetractCoil , PT := ref_stCyl.stCylinderPara.tOriginDebounceTime );
		ref_stCyl.bOriginConfirmed	:= _tonORIDeb.Q ;		
	END_IF
//自動關閉 
	IF ref_stCyl.stCylinderPara.bCoilAutoOff THEN
		IF ref_stCyl.iEndSensor	THEN
			ref_stCyl.qExtendCoil :=FALSE;
		END_IF
		IF ref_stCyl.iOriginSensor	THEN
			ref_stCyl.qRetractCoil :=FALSE;
		END_IF	
	
	END_IF
END_METHOD

METHOD Home : BOOL
VAR_INPUT
END_VAR
CASE ref_stCyl.stCylinderPara.eCylinderType OF 
	E_CylinderType.ThreePort_TwoPosition:
		ref_stCyl.qExtendCoil	:=FALSE;
	E_CylinderType.FivePort_TwoPosition:
		ref_stCyl.qExtendCoil	:=FALSE;
		ref_stCyl.qRetractCoil	:= TRUE;
END_CASE
Home:= ref_stCyl.iOriginSensor;
END_METHOD

METHOD Reset
VAR_INPUT
END_VAR
// ======================================================
//  Reset  — 復歸：清錯 + 停止所有監看/定時器
// ======================================================
(*
// 停止監看
_watchOri := FALSE;
_watchEnd := FALSE;

// 關閉所有 TON
_tonTO_Ori(IN := FALSE);
_tonTO_End(IN := FALSE);
_tonOriDeb(IN := FALSE);
_tonEndDeb(IN := FALSE);
_cc_tonStuck(IN := FALSE);

*)
// 清除錯誤/故障碼
ref_stCyl.eCylFault      := E_CylFault.None;
ref_stCyl.bError         := FALSE;

// （可選）清除已確認狀態，讓到位需重新經過除抖
ref_stCyl.bOriginConfirmed := FALSE;
ref_stCyl.bEndConfirmed    := FALSE;
END_METHOD

METHOD INTERNAL ThreePort_TwoPosition
VAR_INPUT
END_VAR
//異常感測時間	
	_tonTimeOutEnd(IN := ref_stCyl.qExtendCoil AND NOT ref_stCyl.iEndSensor, PT := ref_stCyl.stCylinderPara.tEndTimeout);
	
	IF _tonTimeOutEnd.Q AND NOT ref_stCyl.stCylinderPara.bEndNoSensor THEN		//確認TimeOut + NO Sensor 
		ref_stCyl.eCylFault := E_CylFault.TimeoutExtend;
	END_IF

	_tonTimeOutORI(IN := NOT ref_stCyl.qExtendCoil AND NOT ref_stCyl.iOriginSensor, PT := ref_stCyl.stCylinderPara.tOriginTimeout);
	
	IF _tonTimeOutORI.Q AND NOT ref_stCyl.stCylinderPara.bOriginNoSensor THEN		//確認TimeOut + NO Sensor 
		ref_stCyl.eCylFault := E_CylFault.TimeoutRetract;
	END_IF	

	
//穩定時間 輸出監控 
	
	IF NOT ref_stCyl.stCylinderPara.bEndNoSensor  THEN			//有感測器 
		_tonEndDeb(IN:=ref_stCyl.iEndSensor , PT := ref_stCyl.stCylinderPara.tEndDebounceTime );
		ref_stCyl.bEndConfirmed	:= _tonEndDeb.Q ;
	ELSE														//沒感測器 
		_tonEndDeb(IN:=ref_stCyl.qExtendCoil , PT := ref_stCyl.stCylinderPara.tEndDebounceTime );
		ref_stCyl.bEndConfirmed	:= _tonEndDeb.Q ;		
	END_IF

	
//穩定時間 回歸

	IF NOT ref_stCyl.stCylinderPara.bOriginNoSensor  THEN			//有感測器 
		_tonORIDeb(IN:=ref_stCyl.iOriginSensor , PT := ref_stCyl.stCylinderPara.tOriginDebounceTime );
		ref_stCyl.bOriginConfirmed	:= _tonORIDeb.Q ;
	ELSE														//沒感測器  
		_tonORIDeb(IN:=NOT ref_stCyl.qExtendCoil , PT := ref_stCyl.stCylinderPara.tOriginDebounceTime );
		ref_stCyl.bOriginConfirmed	:= _tonORIDeb.Q ;		
	END_IF
END_METHOD

END_FUNCTION_BLOCK

// ---- 02_Unit/03_Axis/AXIS_REF_Ext.TcPOU
FUNCTION_BLOCK AXIS_REF_Ext EXTENDS AXIS_REF
VAR_INPUT
	EMG					:BOOL;
	Enable_Positive		:BOOL;
	Enable_Negative		:BOOL;
	AxisName			:STRING(50);
END_VAR
VAR_OUTPUT
	strAxisStates		:STRING(50);
	DI					AT %I* :UDINT;
	DeviceErrorcode			AT %I* :WORD;
END_VAR
VAR
	stEcSlaveAmsNetAdr 	AT %I* 			:ST_AmsAddr;
	_IndexCounter						:UDINT;
	MC_Power							:MC_Power;
	MC_Jog								:MC_Jog;
	_bSwich								:BOOL;
	_bJogFFlag,_bJogBFlag,_bStopFlag,_bResetFlag,_bMoveVelocityFlag,_bSetPosition			:BOOL;			//內部旗標 
	MC_Stop								:MC_Stop;
	MC_Reset							:MC_Reset;		
	MC_ReadParameter					:MC_ReadParameter;
	MC_ReadDriveAddress					:MC_ReadDriveAddress;
	MC_MoveVelocity						:MC_MoveVelocity;
	MC_SetPosition						:MC_SetPosition;
	MaxVelo								:LREAL;
	TempVelo							:LREAL;
	nJogStep,nStopStep,nResetStep,nMoveVelocityStep,nSetPositionStep		:INT;
	
	
	
END_VAR

SUPER^.ReadStatus();
SUPER^();
//flagtoString
AxisStatesToString();
/////////////////////////////////Power ON///////////////////////////////////
IF NOT EMG THEN
	_bSwich:=FALSE;
END_IF
MC_Power(
	Axis:= SUPER^, 
	Enable:= _bSwich, 
	Enable_Positive:= Enable_Positive, 
	Enable_Negative:= Enable_Negative, 
	Override:= , 
	BufferMode:= , 
	Options:= , 
	Status=> , 
	Busy=> , 
	Error=> , 
	ErrorID=> );
	
MC_ReadDriveAddress(
	Axis:= SUPER^, 
	Execute:= MC_Power.Status, 
	Done=> , 
	Busy=> , 
	Error=> , 
	ErrorID=> , 
	DriveAddress=> );	
	

///////////////////////////////////////////////////////////////
NStep();

ACTION AxisStatesToString:
CASE SUPER^.Status.MotionState OF
    MC_AXISSTATE_UNDEFINED:
		strAxisStates:='Undefined';
    MC_AXISSTATE_DISABLED:
		strAxisStates:='Disable';
    MC_AXISSTATE_STANDSTILL:
		strAxisStates:='Standstill';
    MC_AXISSTATE_ERRORSTOP:
		strAxisStates:='ErrorStop';
    MC_AXISSTATE_STOPPING:
		strAxisStates:='Stopping';
    MC_AXISSTATE_HOMING:
		strAxisStates:='Homing';
    MC_AXISSTATE_DISCRETEMOTION:
		strAxisStates:='Discretemotion';
    MC_AXISSTATE_CONTINOUSMOTION:
		strAxisStates:='Continousmotion';
    MC_AXISSTATE_SYNCHRONIZEDMOTION	:
		strAxisStates:='Synchronizedmotion';	
END_CASE
END_ACTION

PROPERTY CommandError : BOOL
GET
VAR
END_VAR
VAR_OUTPUT
	ErrorID	:	UDINT;
END_VAR
CommandError:= 	MC_Stop.Error OR MC_Reset.Error OR MC_Jog.Error OR MC_Power.Error OR MC_SetPosition.Error OR MC_MoveVelocity.Error;

ErrorID:=	MC_Stop.ErrorID OR MC_Reset.ErrorID OR MC_Jog.ErrorID OR MC_Power.ErrorID OR MC_SetPosition.ErrorID OR MC_MoveVelocity.ErrorID;
END_GET
END_PROPERTY

PROPERTY Error : BOOL
GET
Error:= SUPER^.Status.Error	OR  SUPER^.Status.DriveDeviceError;
END_GET
END_PROPERTY

METHOD JogBackwards : BOOL
VAR_INPUT
	Velocity: LREAL;
END_VAR
_bJogBFlag	:= TRUE;

IF NOT MC_Jog.JogForward THEN
	IF 	Velocity > MaxVelo THEN
		MC_Jog.Velocity	:= MaxVelo ; 
		ELSE
		MC_Jog.Velocity	:=	Velocity;
	END_IF
END_IF
JogBackwards:= SUPER^.Status.ConstantVelocity;
END_METHOD

METHOD JogForward : BOOL
VAR_INPUT
	Velocity	:LREAL;
END_VAR
_bJogFFlag	:= TRUE;

IF NOT MC_Jog.JogBackwards THEN
	IF 	Velocity > MaxVelo THEN
		MC_Jog.Velocity	:= MaxVelo ; 
		ELSE
		MC_Jog.Velocity	:=	Velocity;
	END_IF
END_IF
JogForward:= SUPER^.Status.ConstantVelocity;
END_METHOD

METHOD MoveVelocity : BOOL
VAR_INPUT
	Velocity			:LREAL;
	Direction 			:TC2_MC2.MC_Direction	 ;
(*MC_Positive_Direction := 1,MC_Shortest_Way ,MC_Negative_Direction,MC_Current_Direction,MC_Undefined_Direction := 128*)	
END_VAR
_bMoveVelocityFlag := TRUE;
TempVelo	:= Velocity ;
MC_MoveVelocity.Direction	:=  Direction;


MoveVelocity:= MC_MoveVelocity.InVelocity;
END_METHOD

ACTION NStep:
//////////////////////////////JOG//////////////////////////////////////	
MC_ReadParameter(
	Axis:= SUPER^, 
	Enable:=TRUE , 
	ParameterNumber:= MaxVelocitySystem, 
	ReadMode:=READMODE_CYCLIC , 
	Valid=> , 
	Busy=> , 
	Error=> , 
	ErrorID=> , 
	Value=> MaxVelo);
////////////////JOG+++//////////////////
MC_Jog(
	Axis:= SUPER^, 
	JogForward:= , 
	JogBackwards:= , 
	Mode:= MC_JOGMODE_CONTINOUS, 
	Position:= , 
	Velocity:= , 
	Acceleration:= , 
	Deceleration:= , 
	Jerk:= , 
	Done=> , 
	Busy=> , 
	Active=> , 
	CommandAborted=> , 
	Error=> , 
	ErrorID=> );
	
IF SUPER^.Status.Error THEN
	nJogStep:=0;
	_bJogFFlag:=FALSE;
	_bJogBFlag:=FALSE;
END_IF	
	
CASE nJogStep OF
	0:
		IF _bJogFFlag THEN
			IF SUPER^.Status.StandStill THEN
				nJogStep:= 10;
			END_IF;
		END_IF
		IF _bJogBFlag THEN
			IF SUPER^.Status.StandStill THEN
				nJogStep:= 15;
			END_IF;
		END_IF		
		
	10:
		MC_Jog.JogForward:=TRUE;
		IF NOT _bJogFFlag THEN
			MC_Jog.JogForward:=FALSE;
			nJogStep:= 0;
		END_IF	
		IF  SUPER^.Status.Stopping THEN
			MC_Jog.JogForward:=FALSE;
			nJogStep:= 20;		
		END_IF
		
	15:
		MC_Jog.JogBackwards:=TRUE;
		IF NOT _bJogBFlag THEN
			MC_Jog.JogBackwards:=FALSE;
			nJogStep:= 0;
		END_IF				
		IF  SUPER^.Status.Stopping THEN
			MC_Jog.JogBackwards:=FALSE;
			nJogStep:=20;		
		END_IF	
	20:
		IF NOT _bJogBFlag AND NOT _bJogFFlag THEN
			nJogStep:= 0;
		END_IF;
	
	50:
END_CASE	

	
_bJogFFlag:=FALSE;
_bJogBFlag:=FALSE;
//********************************************************
//STOP

MC_Stop(
	Axis:=SUPER^ , 
	Execute:= , 
	Deceleration:= , 
	Jerk:= , 
	Options:= , 
	Done=> , 
	Busy=> , 
	Active=> , 
	CommandAborted=> , 
	Error=> , 
	ErrorID=> );
CASE nStopStep OF
	0:	
		MC_Stop.Execute:= FALSE;
		IF _bStopFlag THEN
			MC_Stop.Execute:= TRUE;
			nStopStep	:= 10;	
		END_IF
	10:
		IF MC_Stop.Done THEN
			MC_Stop.Execute:= FALSE;
			nStopStep	:= 15;		
		END_IF;		
		IF MC_Stop.Error THEN
			MC_Stop.Execute:= FALSE;
			nStopStep	:= 20;		
		END_IF;	

		
	15:		
		IF NOT _bStopFlag THEN
			MC_Stop.Execute:= FALSE;
			nStopStep	:= 0;	
		END_IF	
	20:
		IF NOT _bStopFlag THEN
			MC_Stop.Execute:= FALSE;
			nStopStep	:= 0;	
		END_IF		
END_CASE;

_bStopFlag:=FALSE;
////////////////////////////////////////////////////
MC_Reset(Axis:=SUPER^);


CASE nResetStep OF
	0:	
		MC_Reset.Execute:= FALSE;
		IF _bResetFlag THEN
			MC_Reset.Execute:= TRUE;
			nResetStep	:= 10;	
		END_IF
	10:
		IF MC_Reset.Done THEN
			MC_Reset.Execute:= FALSE;
			nResetStep	:= 15;		
		END_IF;		
		IF MC_Reset.Error THEN
			MC_Reset.Execute:= FALSE;
			nResetStep	:= 20;		
		END_IF;	

		
	15:		
		IF NOT _bResetFlag THEN
			nResetStep	:= 0;	
		END_IF	
	20:
		IF NOT _bResetFlag THEN
			nResetStep	:= 0;	
		END_IF	
	
END_CASE;


	
_bResetFlag	:=FALSE;
////////////////////////////////////////////////////////////////////	
MC_MoveVelocity(Axis:= SUPER^);
IF SUPER^.Status.Error  THEN
	nMoveVelocityStep	:= 0;
END_IF

CASE nMoveVelocityStep OF
	0:	
		MC_MoveVelocity.Execute:= FALSE;
		IF _bMoveVelocityFlag AND SUPER^.Status.StandStill AND NOT SUPER^.Status.Error  THEN
			MC_MoveVelocity.Velocity	:= TempVelo;
			MC_MoveVelocity.Execute:= TRUE;
			nMoveVelocityStep	:= 5;
		END_IF
	
	5:
		IF MC_MoveVelocity.Velocity	<> TempVelo THEN
			MC_MoveVelocity.Execute:= FALSE;
			nMoveVelocityStep	:= 6;
		END_IF
		IF NOT _bMoveVelocityFlag THEN
			nMoveVelocityStep	:= 20;
		END_IF
	6:
		IF NOT MC_MoveVelocity.Active THEN
			MC_MoveVelocity.Velocity	:= TempVelo;
			MC_MoveVelocity.Execute		:= TRUE;
			nMoveVelocityStep			:= 5;
		END_IF;		

	20:
		IF Stop() THEN
			nMoveVelocityStep	:= 0;
		END_IF		
	
END_CASE;	
_bMoveVelocityFlag := FALSE;

//////////////////////////////////////////////////////////////
MC_SetPosition(Axis:= SUPER^);
CASE nSetPositionStep OF
	0:
		MC_SetPosition.Execute:= FALSE;
		IF _bSetPosition THEN
			MC_SetPosition.Execute:= TRUE;
			nSetPositionStep:= 5;
		END_IF
	
	5:
		IF MC_SetPosition.Done THEN
			nSetPositionStep:= 10;
		END_IF
		IF MC_SetPosition.Error THEN
			nSetPositionStep:= 15;
		END_IF
	10:
		IF NOT _bSetPosition THEN
			MC_SetPosition.Execute:= FALSE;
			nSetPositionStep:= 0;
		END_IF
	15:
		IF NOT _bSetPosition THEN
			MC_SetPosition.Execute:= FALSE;
			nSetPositionStep:= 0;
		END_IF

END_CASE






_bSetPosition	:=FALSE;
END_ACTION

METHOD Reset : BOOL
VAR_INPUT
END_VAR
_bResetFlag	:=TRUE;
Reset := nResetStep = 15;
END_METHOD

METHOD ServoOFF : BOOL
VAR_INPUT
END_VAR
_bSwich	:= FALSE;
ServoOFF	:= SUPER^.Status.Disabled;
END_METHOD

METHOD ServoOn : BOOL
VAR_INPUT
END_VAR
IF EMG THEN
	_bSwich	:= TRUE;
	ELSE
	_bSwich	:= FALSE;
END_IF
ServoOn := MC_Power.Status;
END_METHOD

METHOD SetPosition : BOOL
VAR_INPUT
	Position:LREAL;
END_VAR
_bSetPosition	:=TRUE;
MC_SetPosition.Position:= Position;

SetPosition	:= MC_SetPosition.Done;
END_METHOD

METHOD Stop : BOOL
VAR_INPUT
END_VAR
_bStopFlag	:= TRUE;
Stop:=  nStopStep=15 ;
END_METHOD

END_FUNCTION_BLOCK

// ---- 02_Unit/01_Customization/Ass_StackComv.TcPOU
FUNCTION_BLOCK Ass_StackComv IMPLEMENTS ITF_AutoStructCommand
VAR_INPUT
END_VAR
VAR_OUTPUT
END_VAR
VAR
	strText	:STRING;
	i	:INT;
	_bProcessScan,_bInitialScan: BOOL;
	_bHalt , _bError,_bHaltPause: BOOL;
	nStep,nInitiStep  	: INT;
	_tmrT0,_tmrT1		:TON;
	bBoxPass: BOOL;
END_VAR

IF NOT _bInitialScan THEN
	nInitiStep	:= 0;
END_IF

_bInitialScan:=FALSE;



IF NOT _bProcessScan THEN
	nStep	:= 0;
END_IF

_bProcessScan:=FALSE;

{warning 'add property implementation'}
PROPERTY Connect : STRING(50)
GET
END_GET
SET
END_SET
END_PROPERTY

{warning 'add property implementation'}
PROPERTY Error : BOOL
GET
END_GET
END_PROPERTY

{warning 'add method implementation '}
METHOD ErrorClear : BOOL
END_METHOD

{warning 'add method implementation '}
METHOD FB_init : BOOL
VAR_INPUT
	(* if TRUE, the retain variables are initialized (warm start / cold start)*)
	bInitRetains	: BOOL;
	(* if TRUE, the instance afterwards gets moved into the copy code (online change)*)
	bInCopyCode	: BOOL;
END_VAR
END_METHOD

{warning 'add method implementation '}
METHOD HaltStepContiune : BOOL
END_METHOD

METHOD Initialization : BOOL
VAR_INPUT
	_Testmode	: BOOL;
END_VAR
_bInitialScan:=TRUE;

CASE nInitiStep OF
	0:		
		strText					:= 'ORG : Inital';
		Motor_Stack.qRun		:=FALSE;
		Vacm_StackUD			:=FALSE;
		Cyl_StackUD.qExtendCoil	:=FALSE;
		Bundling_yPause			:= FALSE;	
		nInitiStep				:= 5;	
	5:
		IF 	Cyl_StackUD.iOriginSensor THEN
			nInitiStep				:= 10;	
		END_IF;
	10:
			strText:='ORG : Done ';
			Initialization	:= TRUE;
	
END_CASE;
END_METHOD

{warning 'add property implementation'}
PROPERTY NoEntry : BOOL
GET
END_GET
END_PROPERTY

{warning 'add method implementation '}
METHOD Pause : BOOL
END_METHOD

METHOD Process : BOOL
VAR_INPUT
	bHlatMode	: BOOL;
END_VAR
_bProcessScan	:= TRUE;
CASE nStep OF 
	0:
		Vacm_StackUD			:=FALSE;
		Cyl_StackUD.qExtendCoil	:=FALSE;
		Motor_Stack.qRun		:=TRUE;
		nStep					:= 5;
		_tmrT0(IN:=FALSE);
		_tmrT1(IN:=FALSE);
	5:
		IF RunParameter.stack_bUsed THEN
				IF Sen_StackComvStop THEN
					Motor_Stack.qRun		:=FALSE;
					nStep					:= 9;
				END_IF
			ELSE		
		
			;
		
		
		END_IF
	9:
		_tmrT0(IN:=TRUE,PT:=T#1S);
		IF _tmrT0.Q THEN
			_tmrT0(IN:=FALSE);
			nStep					:= 10;
		END_IF		
		
	10://堆疊1
		Cyl_StackUD.qExtendCoil	:= TRUE;
		_tmrT0(IN:=TRUE,PT:=RunParameter.stack_DelayTime1);
		IF _tmrT0.Q THEN
			_tmrT0(IN:=FALSE);
			nStep					:= 15;
		END_IF
	15:
		Vacm_StackUD			:=TRUE;	
		_tmrT0(IN:=TRUE,PT:=T#1S);
		IF _tmrT0.Q THEN
			_tmrT0(IN:=FALSE);
			nStep					:= 20;
		END_IF
	20:
		Cyl_StackUD.qExtendCoil	:= FALSE;		
		IF Cyl_StackUD.iOriginSensor THEN
			nStep					:= 25;
		END_IF		
	25:
		Motor_Stack.qRun		:=TRUE;
		IF Sen_StackComvStop THEN
			Motor_Stack.qRun		:=FALSE;
			nStep					:= 30;
		END_IF	
	30:	
		_tmrT0(IN:=TRUE,PT:=T#1S);
		IF _tmrT0.Q THEN
			_tmrT0(IN:=FALSE);
			nStep					:= 35;
		END_IF		
	
	35:		
		Cyl_StackUD.qExtendCoil	:= TRUE;
		_tmrT0(IN:=TRUE,PT:=RunParameter.stack_DelayTime2);
		IF _tmrT0.Q THEN
			_tmrT0(IN:=FALSE);
			nStep					:= 40;
		END_IF		
	40:
		Cyl_StackUD.qExtendCoil	:= FALSE;
		Vacm_StackUD			:=FALSE;
		_tmrT0(IN:=TRUE,PT:=T#0.5S);
		IF _tmrT0.Q THEN
			_tmrT0(IN:=FALSE);
			nStep					:= 45;
		END_IF						
	45:
		Motor_Stack.qRun		:=TRUE;
		IF NOT Sen_StackComvStop THEN
			nStep					:=0;
		END_IF	
	
	
	
	
END_CASE
END_METHOD

{warning 'add property implementation'}
PROPERTY Status : STRING(50)
GET
END_GET
END_PROPERTY

END_FUNCTION_BLOCK

// ---- 02_Unit/01_Customization/Ass_Sealing.TcPOU
FUNCTION_BLOCK Ass_Sealing IMPLEMENTS ITF_AutoStructCommand
VAR_INPUT
END_VAR
VAR_OUTPUT
END_VAR
VAR
	i	:INT;
	_bProcessScan,_bInitialScan: BOOL;
	_bHalt , _bError,_bHaltPause: BOOL;
	strText	:STRING;
	nStep,nInitiStep ,nNextStep 	: INT;
	_tmrT0			:TON;
END_VAR

IF NOT _bInitialScan THEN
	nInitiStep	:= 0;
END_IF

_bInitialScan:=FALSE;



IF NOT _bProcessScan THEN
	nNextStep	:= 0;
	nStep		:= 0;
END_IF

_bProcessScan	:=FALSE;

PROPERTY Connect : STRING(50)
GET
CASE nStep OF
	5:
	Connect	:= 'OpenBox In';
	20:
	Connect	:= 'Ready'; 
	50:
	Connect	:= 'LoadPic In';
	ELSE	
	Connect	:= '';		
END_CASE
END_GET
SET
END_SET
END_PROPERTY

{warning 'add property implementation'}
PROPERTY Error : BOOL
GET
END_GET
END_PROPERTY

{warning 'add method implementation '}
METHOD ErrorClear : BOOL
END_METHOD

{warning 'add method implementation '}
METHOD FB_init : BOOL
VAR_INPUT
	(* if TRUE, the retain variables are initialized (warm start / cold start)*)
	bInitRetains	: BOOL;
	(* if TRUE, the instance afterwards gets moved into the copy code (online change)*)
	bInCopyCode	: BOOL;
END_VAR
END_METHOD

{warning 'add method implementation '}
METHOD HaltStepContiune : BOOL
END_METHOD

METHOD Initialization : BOOL
VAR_INPUT
	_Testmode	: BOOL;
END_VAR

VAR
	bConfig: BOOL;
END_VAR
_bInitialScan:=TRUE;

CASE nInitiStep OF
	0:		
		_tmrT0(IN:=FALSE);
		strText:='ORG : Initial ';
		Motor_BoxSealBottom_L.qRun		:=FALSE;
		Motor_BoxSealBottom_R.qRun		:=FALSE;
		Cyl_BeltBottomSup.qExtendCoil	:=FALSE;		
		nInitiStep						:= 5;
	5:
	bConfig			:=TRUE;
	IF Sen_BeltLoadIn OR Sen_BeltLoadOut THEN
		bConfig			:=FALSE;
		EventLogger.eEventType		:= 4;
		EventLogger.strEventText	:= 'Sensor Error ';	
		EventLogger();					
	END_IF		
	IF NOT Motor_BoxSealBottom_R.iError OR NOT Motor_BoxSealBottom_L.iError  THEN
		bConfig			:=FALSE;
		EventLogger.eEventType		:= 4;
		EventLogger.strEventText	:= 'INV. Motor Error ';	
		EventLogger();					
	END_IF	
	
	IF bConfig THEN
		strText:='ORG : Done ';
		nInitiStep	:= 20;
		ELSE
		strText:='ORG : Failed ';
		nInitiStep	:= 50;
	END_IF
	
	
	
	
	

20:
	Initialization	:= TRUE;

END_CASE;
END_METHOD

{warning 'add property implementation'}
PROPERTY NoEntry : BOOL
GET
END_GET
END_PROPERTY

{warning 'add method implementation '}
METHOD Pause : BOOL
END_METHOD

METHOD Process : BOOL
VAR_INPUT
	bHlatMode	: BOOL;
END_VAR


_bProcessScan	:= TRUE;
//判斷 

IF _bError THEN
	strText	:= 'OpenBox:Error ';
	strText	:= CONCAT(Status,INT_TO_STRING(nStep));
END_IF;
//半自動模式
IF NOT bHlatMode  THEN
	nStep:= nNextStep;	
END_IF;

_bHaltPause	:= nStep<> nNextStep;
IF _bError OR _bHaltPause THEN
	RETURN;
END_IF

//主程序 
IF NOT _bHaltPause THEN
	CASE nStep OF
		0:
			_tmrT0(IN:=FALSE);
			Motor_BoxSealBottom_L.qRun		:=TRUE;
			Motor_BoxSealBottom_R.qRun		:=TRUE;
			nNextStep						:= 5;
			strText							:= 'Waiting for load';
		5:
			IF Sen_BeltLoadIn THEN
				Cyl_BeltBottomSup.qExtendCoil	:=TRUE;
				strText							:= 'load In';
				nNextStep						:= 10;
			END_IF;	
		10:
			IF NOT Sen_BeltLoadIn THEN
				//Cyl_BeltBottomSup.qExtendCoil	:=FALSE;
				;
			END_IF;		
	
			IF Sen_BeltLoadOut THEN
				Cyl_BeltBottomSup.qExtendCoil	:=FALSE;
				strText						:= 'load Out';
				nNextStep					:= 15;
			END_IF;		
		15:
			_tmrT0(IN:=TRUE,PT:=T#0.5S);
			IF _tmrT0.Q THEN
				_tmrT0(IN:=FALSE);
				IF OP.xAutoMode THEN
					nNextStep					:= 20;
					ELSE
					nNextStep					:= 50;
				END_IF;
			END_IF
		20:
				IF M_LoadPic3.Connect= 'Seal In' THEN
					nNextStep					:= 21;
					ELSE
					Motor_BoxSealBottom_L.qRun		:=FALSE;
					Motor_BoxSealBottom_R.qRun		:=FALSE;
				END_IF
		21:
				_tmrT0(IN:=NOT Sen_BeltLoadOut,PT:=T#0.5S);
				Motor_BoxSealBottom_L.qRun		:=TRUE;
				Motor_BoxSealBottom_R.qRun		:=TRUE;		
				IF 	_tmrT0.Q THEN
					_tmrT0(IN:=FALSE);
					nNextStep					:= 50;
				END_IF
		50:
				nNextStep					:= 0;
	END_CASE
END_IF;

Process	:= nStep =50;
END_METHOD

{warning 'add property implementation'}
PROPERTY Status : STRING(50)
GET
END_GET
END_PROPERTY

END_FUNCTION_BLOCK

// ---- 02_Unit/01_Customization/Ass_UnloadNG.TcPOU
FUNCTION_BLOCK Ass_UnloadNG IMPLEMENTS ITF_AutoStructCommand
VAR_INPUT
END_VAR
VAR_OUTPUT
	SamplingWeight	:REAL;
END_VAR
VAR
	strText,strNGText,strShackText 	:STRING;
	i	:INT;
	_bProcessScan,_bInitialScan: BOOL;
	_bHalt , _bError,_bHaltPause: BOOL;
	nStep,nInitiStep ,nNGStep,nShackStep 	: INT;
	_tmrT0,tmrLoadcell,tmrshock	,tmrNG		:TON;
	bBoxPass: BOOL;
	tmrClear: TON;
	UpperWeight,LowerWeight	:REAL;
END_VAR

IF NOT _bInitialScan AND NOT _bProcessScan THEN
	strText:=strNGText:=strShackText	:='';
END_IF


IF NOT _bInitialScan THEN
	nInitiStep	:= 0;
END_IF

_bInitialScan:=FALSE;



IF NOT _bProcessScan THEN
	nShackStep	:= 0;
	nNGStep		:= 0;
	nStep		:= 0;
END_IF

_bProcessScan	:=FALSE;

{warning 'add property implementation'}
PROPERTY Connect : STRING(50)
GET
END_GET
SET
END_SET
END_PROPERTY

PROPERTY Error : BOOL
GET
END_GET
END_PROPERTY

METHOD ErrorClear : BOOL
_bError	:= FALSE;
END_METHOD

{warning 'add method implementation '}
METHOD FB_init : BOOL
VAR_INPUT
	(* if TRUE, the retain variables are initialized (warm start / cold start)*)
	bInitRetains	: BOOL;
	(* if TRUE, the instance afterwards gets moved into the copy code (online change)*)
	bInCopyCode	: BOOL;
END_VAR
END_METHOD

METHOD HaltStepContiune : BOOL
HaltStepContiune	:=TRUE;
END_METHOD

